LIN {X 0,Y 291.529,Z 647.486,A -85,B 0,C 180,E1 -16988.801,E2 -16988.801} C_VEL
LIN {X 0,Y 290.055,Z 656.21,A -85,B 0,C 180,E1 -16989.986,E2 -16989.986} C_VEL
LIN {X 0,Y 288.759,Z 663.631,A -85,B 0,C 180,E1 -16991.187,E2 -16991.187} C_VEL
LIN {X 0,Y 287.31,Z 672.431,A -85,B 0,C 180,E1 -16992.93,E2 -16992.93} C_VEL
LIN {X 0,Y 286.152,Z 678.42,A -85,B 0,C 180,E1 -16994.326,E2 -16994.326} C_VEL
LIN {X 0,Y 284.969,Z 684.732,A -85,B 0,C 180,E1 -16996.087,E2 -16996.087} C_VEL
LIN {X 0,Y 283.972,Z 690.005,A -85,B 0,C 180,E1 -16997.856,E2 -16997.856} C_VEL
LIN {X 0,Y 283.192,Z 695.101,A -85,B 0,C 180,E1 -16999.996,E2 -16999.996} C_VEL
LIN {X 0,Y 282.682,Z 699.069,A -85,B 0,C 180,E1 -17002.141,E2 -17002.141} C_VEL
LIN {X 0,Y 282.337,Z 702.443,A -85,B 0,C 180,E1 -17004.694,E2 -17004.694} C_VEL
LIN {X 0,Y 282.309,Z 703.508,A -85,B 0,C 180,E1 -17005.717,E2 -17005.717} C_VEL
LIN {X 0,Y 282.334,Z 705.035,A -85,B 0,C 180,E1 -17008.574,E2 -17008.574} C_VEL
LIN {X 0,Y 282.347,Z 705.315,A -85,B 0,C 180,E1 -17010,E2 -17010} C_VEL
LIN {X 0,Y 282.339,Z 704.439,A -85,B 0,C 180,E1 -17012.854,E2 -17012.854} C_VEL
LIN {X 0,Y 282.309,Z 703.508,A -85,B 0,C 180,E1 -17014.283,E2 -17014.283} C_VEL
LIN {X 0,Y 282.523,Z 700.157,A -85,B 0,C 180,E1 -17017.145,E2 -17017.145} C_VEL
LIN {X 0,Y 282.991,Z 696.53,A -85,B 0,C 180,E1 -17019.29,E2 -17019.29} C_VEL
LIN {X 0,Y 283.711,Z 691.797,A -85,B 0,C 180,E1 -17021.43,E2 -17021.43} C_VEL
LIN {X 0,Y 284.732,Z 685.823,A -85,B 0,C 180,E1 -17023.561,E2 -17023.561} C_VEL
LIN {X 0,Y 285.91,Z 679.733,A -85,B 0,C 180,E1 -17025.322,E2 -17025.322} C_VEL
LIN {X 0,Y 287.02,Z 673.992,A -85,B 0,C 180,E1 -17026.721,E2 -17026.721} C_VEL
LIN {X 0,Y 288.238,Z 667.091,A -85,B 0,C 180,E1 -17028.16,E2 -17028.16} C_VEL
LIN {X 0,Y 289.495,Z 659.505,A -85,B 0,C 180,E1 -17029.5,E2 -17029.5} C_VEL
LIN {X 0,Y 290.886,Z 651.424,A -85,B 0,C 180,E1 -17030.692,E2 -17030.692} C_VEL
LIN {X 0,Y 292.442,Z 641.666,A -85,B 0,C 180,E1 -17031.869,E2 -17031.869} C_VEL
LIN {X 0,Y 293.596,Z 633.277,A -85,B 0,C 180,E1 -17032.705,E2 -17032.705} C_VEL
LIN {X 0,Y 294.808,Z 622.772,A -85,B 0,C 180,E1 -17033.535,E2 -17033.535} C_VEL
LIN {X 0,Y 295.738,Z 612.44,A -85,B 0,C 180,E1 -17034.154,E2 -17034.154} C_VEL
LIN {X 0,Y 296.591,Z 601.726,A -85,B 0,C 180,E1 -17034.592,E2 -17034.592} C_VEL
LIN {X 0,Y 297.298,Z 578.95,A -85,B 0,C 180,E1 -17035.183,E2 -17035.183} C_VEL
LIN {X 0,Y 298.186,Z 540.495,A -85,B 0,C 180,E1 -17036.108,E2 -17036.108} C_VEL
LIN {X 0,Y 294.791,Z 520.737,A -85,B 0,C 180,E1 -17036.956,E2 -17036.956} C_VEL
LIN {X 0,Y 290.227,Z 500.059,A -85,B 0,C 180,E1 -17037.976,E2 -17037.976} C_VEL
LIN {X 0,Y 288.063,Z 494.317,A -85,B 0,C 180,E1 -17038.404,E2 -17038.404} C_VEL
LIN {X 0,Y 287.664,Z 492.009,A -85,B 0,C 180,E1 -17039.25,E2 -17039.25} C_VEL
LIN {X 0,Y 286.155,Z 484.135,A -85,B 0,C 180,E1 -17042.705,E2 -17042.705} C_VEL
LIN {X 0,Y 284.354,Z 475.643,A -85,B 0,C 180,E1 -17046.602,E2 -17046.602} C_VEL
LIN {X 0,Y 284.259,Z 475.55,A -85,B 0,C 180,E1 -17050.002,E2 -17050.002} C_VEL
LIN {X 0,Y 284.237,Z 475.58,A -85,B 0,C 180,E1 -17054.186,E2 -17054.186} C_VEL
LIN {X 0,Y 284.242,Z 475.579,A -85,B 0,C 180,E1 -17058.117,E2 -17058.117} C_VEL
LIN {X 0,Y 284.297,Z 475.566,A -85,B 0,C 180,E1 -17061.827,E2 -17061.827} C_VEL
LIN {X 0,Y 284.309,Z 475.551,A -85,B 0,C 180,E1 -17065.349,E2 -17065.349} C_VEL
LIN {X 0,Y 284.287,Z 475.573,A -85,B 0,C 180,E1 -17068.723,E2 -17068.723} C_VEL
LIN {X 0,Y 284.275,Z 475.553,A -85,B 0,C 180,E1 -17071.981,E2 -17071.981} C_VEL
LIN {X 0,Y 284.293,Z 475.566,A -85,B 0,C 180,E1 -17076.158,E2 -17076.158} C_VEL
LIN {X 0,Y 284.334,Z 475.543,A -85,B 0,C 180,E1 -17079.926,E2 -17079.926} C_VEL
LIN {X 0,Y 284.419,Z 475.547,A -85,B 0,C 180,E1 -17084.51,E2 -17084.51} C_VEL
LIN {X 0,Y 284.45,Z 475.533,A -85,B 0,C 180,E1 -17088.598,E2 -17088.598} C_VEL
LIN {X 0,Y 284.578,Z 475.499,A -85,B 0,C 180,E1 -17091.477,E2 -17091.477} C_VEL
LIN {X 0,Y 284.562,Z 475.535,A -85,B 0,C 180,E1 -17094.328,E2 -17094.328} C_VEL
LIN {X 0,Y 284.832,Z 475.483,A -85,B 0,C 180,E1 -17098.584,E2 -17098.584} C_VEL
LIN {X 0,Y 284.831,Z 475.469,A -85,B 0,C 180,E1 -17101.412,E2 -17101.412} C_VEL
LIN {X 0,Y 284.636,Z 475.523,A -85,B 0,C 180,E1 -17107.089,E2 -17107.089} C_VEL
LIN {X 0,Y 284.508,Z 475.507,A -85,B 0,C 180,E1 -17109.955,E2 -17109.955} C_VEL
LIN {X 0,Y 284.427,Z 475.557,A -85,B 0,C 180,E1 -17114.303,E2 -17114.303} C_VEL
LIN {X 0,Y 284.305,Z 475.536,A -85,B 0,C 180,E1 -17118.743,E2 -17118.743} C_VEL
LIN {X 0,Y 284.288,Z 475.562,A -85,B 0,C 180,E1 -17121.764,E2 -17121.764} C_VEL
LIN {X 0,Y 284.28,Z 475.569,A -85,B 0,C 180,E1 -17124.849,E2 -17124.849} C_VEL
LIN {X 0,Y 284.255,Z 475.55,A -85,B 0,C 180,E1 -17128.016,E2 -17128.016} C_VEL
LIN {X 0,Y 284.269,Z 475.576,A -85,B 0,C 180,E1 -17131.274,E2 -17131.274} C_VEL
LIN {X 0,Y 284.326,Z 475.549,A -85,B 0,C 180,E1 -17135.345,E2 -17135.345} C_VEL
LIN {X 0,Y 284.253,Z 475.578,A -85,B 0,C 180,E1 -17138.175,E2 -17138.175} C_VEL
LIN {X 0,Y 284.224,Z 475.571,A -85,B 0,C 180,E1 -17142.115,E2 -17142.115} C_VEL
LIN {X 0,Y 284.223,Z 475.543,A -85,B 0,C 180,E1 -17146.184,E2 -17146.184} C_VEL
LIN {X 0,Y 284.243,Z 475.546,A -85,B 0,C 180,E1 -17150.035,E2 -17150.035} C_VEL
LIN {X 0,Y 284.306,Z 475.551,A -85,B 0,C 180,E1 -17153.611,E2 -17153.611} C_VEL
LIN {X 0,Y 284.293,Z 475.554,A -85,B 0,C 180,E1 -17157.189,E2 -17157.189} C_VEL
LIN {X 0,Y 284.294,Z 475.725,A -85,B 0,C 180,E1 -17160.852,E2 -17160.852} C_VEL
LIN {X 0,Y 284.519,Z 476.73,A -85,B 0,C 180,E1 -17161.125,E2 -17161.125} C_VEL
LIN {X 0,Y 292.878,Z 492.327,A -85,B 0,C 180,E1 -17162.476,E2 -17162.476} C_VEL
LIN {X 0,Y 300.917,Z 503.502,A -85,B 0,C 180,E1 -17163.57,E2 -17163.57} C_VEL
LIN {X 0,Y 308.987,Z 512.535,A -85,B 0,C 180,E1 -17164.628,E2 -17164.628} C_VEL
LIN {X 0,Y 315.644,Z 519.573,A -85,B 0,C 180,E1 -17165.615,E2 -17165.615} C_VEL
LIN {X 0,Y 321.421,Z 525.437,A -85,B 0,C 180,E1 -17166.558,E2 -17166.558} C_VEL
LIN {X 0,Y 328.657,Z 532.455,A -85,B 0,C 180,E1 -17167.889,E2 -17167.889} C_VEL
LIN {X 0,Y 335.557,Z 538.982,A -85,B 0,C 180,E1 -17169.296,E2 -17169.296} C_VEL
LIN {X 0,Y 343.686,Z 546.102,A -85,B 0,C 180,E1 -17171.087,E2 -17171.087} C_VEL
LIN {X 0,Y 348.971,Z 550.286,A -85,B 0,C 180,E1 -17172.362,E2 -17172.362} C_VEL
LIN {X 0,Y 354.495,Z 554.841,A -85,B 0,C 180,E1 -17173.83,E2 -17173.83} C_VEL
LIN {X 0,Y 358.656,Z 557.939,A -85,B 0,C 180,E1 -17175.02,E2 -17175.02} C_VEL
LIN {X 0,Y 363.351,Z 561.774,A -85,B 0,C 180,E1 -17176.526,E2 -17176.526} C_VEL
LIN {X 0,Y 367.654,Z 564.654,A -85,B 0,C 180,E1 -17178.042,E2 -17178.042} C_VEL
LIN {X 0,Y 370.229,Z 566.282,A -85,B 0,C 180,E1 -17179.057,E2 -17179.057} C_VEL
LIN {X 0,Y 373.801,Z 569.424,A -85,B 0,C 180,E1 -17180.707,E2 -17180.707} C_VEL
LIN {X 0,Y 376.944,Z 571.542,A -85,B 0,C 180,E1 -17182.409,E2 -17182.409} C_VEL
LIN {X 0,Y 379.734,Z 573.137,A -85,B 0,C 180,E1 -17184.311,E2 -17184.311} C_VEL
LIN {X 0,Y 381.683,Z 573.837,A -85,B 0,C 180,E1 -17186.144,E2 -17186.144} C_VEL
LIN {X 0,Y 382.823,Z 574.391,A -85,B 0,C 180,E1 -17187.896,E2 -17187.896} C_VEL
LIN {X 0,Y 383.197,Z 574.651,A -85,B 0,C 180,E1 -17188.949,E2 -17188.949} C_VEL
LIN {X 0,Y 383.338,Z 574.609,A -85,B 0,C 180,E1 -17190,E2 -17190} C_VEL
LIN {X 0,Y 382.956,Z 574.451,A -85,B 0,C 180,E1 -17191.84,E2 -17191.84} C_VEL
LIN {X 0,Y 381.682,Z 573.849,A -85,B 0,C 180,E1 -17193.854,E2 -17193.854} C_VEL
LIN {X 0,Y 379.685,Z 573.06,A -85,B 0,C 180,E1 -17195.732,E2 -17195.732} C_VEL
LIN {X 0,Y 376.692,Z 571.448,A -85,B 0,C 180,E1 -17197.73,E2 -17197.73} C_VEL
LIN {X 0,Y 373.535,Z 569.224,A -85,B 0,C 180,E1 -17199.421,E2 -17199.421} C_VEL
LIN {X 0,Y 369.66,Z 565.748,A -85,B 0,C 180,E1 -17201.184,E2 -17201.184} C_VEL
LIN {X 0,Y 365.169,Z 563.042,A -85,B 0,C 180,E1 -17202.852,E2 -17202.852} C_VEL
LIN {X 0,Y 360.317,Z 559.407,A -85,B 0,C 180,E1 -17204.458,E2 -17204.458} C_VEL
LIN {X 0,Y 356.054,Z 555.938,A -85,B 0,C 180,E1 -17205.739,E2 -17205.739} C_VEL
LIN {X 0,Y 350.445,Z 551.606,A -85,B 0,C 180,E1 -17207.252,E2 -17207.252} C_VEL
LIN {X 0,Y 345.679,Z 547.625,A -85,B 0,C 180,E1 -17208.44,E2 -17208.44} C_VEL
LIN {X 0,Y 339.714,Z 542.632,A -85,B 0,C 180,E1 -17209.815,E2 -17209.815} C_VEL
LIN {X 0,Y 331.377,Z 535.125,A -85,B 0,C 180,E1 -17211.572,E2 -17211.572} C_VEL
LIN {X 0,Y 323.219,Z 527.28,A -85,B 0,C 180,E1 -17213.117,E2 -17213.117} C_VEL
LIN {X 0,Y 316.382,Z 520.409,A -85,B 0,C 180,E1 -17214.265,E2 -17214.265} C_VEL
LIN {X 0,Y 309.394,Z 512.951,A -85,B 0,C 180,E1 -17215.317,E2 -17215.317} C_VEL
LIN {X 0,Y 301.321,Z 504.014,A -85,B 0,C 180,E1 -17216.378,E2 -17216.378} C_VEL
LIN {X 0,Y 293.463,Z 493.195,A -85,B 0,C 180,E1 -17217.44,E2 -17217.44} C_VEL
LIN {X 0,Y 287.712,Z 482.971,A -85,B 0,C 180,E1 -17218.326,E2 -17218.326} C_VEL
LIN {X 0,Y 284.463,Z 476.5,A -85,B 0,C 180,E1 -17218.907,E2 -17218.907} C_VEL
LIN {X 0,Y 284.265,Z 475.622,A -85,B 0,C 180,E1 -17219.234,E2 -17219.234} C_VEL
LIN {X 0,Y 284.291,Z 475.552,A -85,B 0,C 180,E1 -17222.947,E2 -17222.947} C_VEL
LIN {X 0,Y 284.306,Z 475.551,A -85,B 0,C 180,E1 -17226.389,E2 -17226.389} C_VEL
LIN {X 0,Y 284.242,Z 475.545,A -85,B 0,C 180,E1 -17230.005,E2 -17230.005} C_VEL
LIN {X 0,Y 284.22,Z 475.552,A -85,B 0,C 180,E1 -17234.189,E2 -17234.189} C_VEL
LIN {X 0,Y 284.227,Z 475.569,A -85,B 0,C 180,E1 -17238.12,E2 -17238.12} C_VEL
LIN {X 0,Y 284.271,Z 475.577,A -85,B 0,C 180,E1 -17242.291,E2 -17242.291} C_VEL
LIN {X 0,Y 284.296,Z 475.549,A -85,B 0,C 180,E1 -17245.352,E2 -17245.352} C_VEL
LIN {X 0,Y 284.269,Z 475.576,A -85,B 0,C 180,E1 -17248.726,E2 -17248.726} C_VEL
LIN {X 0,Y 284.255,Z 475.55,A -85,B 0,C 180,E1 -17251.984,E2 -17251.984} C_VEL
LIN {X 0,Y 284.29,Z 475.575,A -85,B 0,C 180,E1 -17256.16,E2 -17256.16} C_VEL
LIN {X 0,Y 284.326,Z 475.536,A -85,B 0,C 180,E1 -17259.93,E2 -17259.93} C_VEL
LIN {X 0,Y 284.408,Z 475.558,A -85,B 0,C 180,E1 -17264.519,E2 -17264.519} C_VEL
LIN {X 0,Y 284.456,Z 475.522,A -85,B 0,C 180,E1 -17268.603,E2 -17268.603} C_VEL
LIN {X 0,Y 284.603,Z 475.509,A -85,B 0,C 180,E1 -17271.482,E2 -17271.482} C_VEL
LIN {X 0,Y 284.56,Z 475.539,A -85,B 0,C 180,E1 -17274.333,E2 -17274.333} C_VEL
LIN {X 0,Y 284.831,Z 475.469,A -85,B 0,C 180,E1 -17278.588,E2 -17278.588} C_VEL
LIN {X 0,Y 284.832,Z 475.483,A -85,B 0,C 180,E1 -17281.416,E2 -17281.416} C_VEL
LIN {X 0,Y 284.634,Z 475.511,A -85,B 0,C 180,E1 -17287.094,E2 -17287.094} C_VEL
LIN {X 0,Y 284.507,Z 475.507,A -85,B 0,C 180,E1 -17289.959,E2 -17289.959} C_VEL
LIN {X 0,Y 284.404,Z 475.555,A -85,B 0,C 180,E1 -17294.309,E2 -17294.309} C_VEL
LIN {X 0,Y 284.326,Z 475.538,A -85,B 0,C 180,E1 -17297.257,E2 -17297.257} C_VEL
LIN {X 0,Y 284.327,Z 475.542,A -85,B 0,C 180,E1 -17299.986,E2 -17299.986} C_VEL
LIN {X 0,Y 283.715,Z 475.635,A -85,B 0,C 180,E1 -17301.168,E2 -17301.168} C_VEL
LIN {X 0,Y 280.834,Z 476,A -85,B 0,C 180,E1 -17303.093,E2 -17303.093} C_VEL
LIN {X 0,Y 278.355,Z 476.3,A -85,B 0,C 180,E1 -17304.657,E2 -17304.657} C_VEL
LIN {X 0,Y 277.296,Z 476.415,A -85,B 0,C 180,E1 -17305.871,E2 -17305.871} C_VEL
LIN {X 0,Y 277.216,Z 476.422,A -85,B 0,C 180,E1 -17306.283,E2 -17306.283} C_VEL
LIN {X 0,Y 277.25,Z 476.449,A -85,B 0,C 180,E1 -17310.475,E2 -17310.475} C_VEL
LIN {X 0,Y 277.248,Z 476.426,A -85,B 0,C 180,E1 -17313.898,E2 -17313.898} C_VEL
LIN {X 0,Y 277.253,Z 476.45,A -85,B 0,C 180,E1 -17317.474,E2 -17317.474} C_VEL
LIN {X 0,Y 277.187,Z 476.454,A -85,B 0,C 180,E1 -17321.243,E2 -17321.243} C_VEL
LIN {X 0,Y 277.177,Z 476.456,A -85,B 0,C 180,E1 -17325.234,E2 -17325.234} C_VEL
LIN {X 0,Y 277.18,Z 476.428,A -85,B 0,C 180,E1 -17328.759,E2 -17328.759} C_VEL
LIN {X 0,Y 277.303,Z 476.579,A -85,B 0,C 180,E1 -17332.849,E2 -17332.849} C_VEL
LIN {X 0,Y 278.891,Z 483.907,A -85,B 0,C 180,E1 -17336.331,E2 -17336.331} C_VEL
LIN {X 0,Y 280.441,Z 491.786,A -85,B 0,C 180,E1 -17339.92,E2 -17339.92} C_VEL
LIN {X 0,Y 280.846,Z 494.095,A -85,B 0,C 180,E1 -17340.795,E2 -17340.795} C_VEL
LIN {X 0,Y 284.507,Z 503.564,A -85,B 0,C 180,E1 -17341.514,E2 -17341.514} C_VEL
LIN {X 0,Y 289.339,Z 526.516,A -85,B 0,C 180,E1 -17342.657,E2 -17342.657} C_VEL
LIN {X 0,Y 291.813,Z 541.536,A -85,B 0,C 180,E1 -17343.311,E2 -17343.311} C_VEL
LIN {X 0,Y 290.242,Z 600.213,A -85,B 0,C 180,E1 -17344.785,E2 -17344.785} C_VEL
LIN {X 0,Y 289.578,Z 609.664,A -85,B 0,C 180,E1 -17345.155,E2 -17345.155} C_VEL
LIN {X 0,Y 288.729,Z 618.789,A -85,B 0,C 180,E1 -17345.652,E2 -17345.652} C_VEL
LIN {X 0,Y 287.555,Z 629.145,A -85,B 0,C 180,E1 -17346.409,E2 -17346.409} C_VEL
LIN {X 0,Y 286.303,Z 638.289,A -85,B 0,C 180,E1 -17347.256,E2 -17347.256} C_VEL
LIN {X 0,Y 284.911,Z 647.289,A -85,B 0,C 180,E1 -17348.284,E2 -17348.284} C_VEL
LIN {X 0,Y 283.4,Z 656.014,A -85,B 0,C 180,E1 -17349.496,E2 -17349.496} C_VEL
LIN {X 0,Y 282.017,Z 663.434,A -85,B 0,C 180,E1 -17350.72,E2 -17350.72} C_VEL
LIN {X 0,Y 280.743,Z 671.058,A -85,B 0,C 180,E1 -17352.235,E2 -17352.235} C_VEL
LIN {X 0,Y 279.28,Z 678.223,A -85,B 0,C 180,E1 -17353.93,E2 -17353.93} C_VEL
LIN {X 0,Y 278.035,Z 684.534,A -85,B 0,C 180,E1 -17355.732,E2 -17355.732} C_VEL
LIN {X 0,Y 276.993,Z 689.807,A -85,B 0,C 180,E1 -17357.546,E2 -17357.546} C_VEL
LIN {X 0,Y 276.181,Z 694.905,A -85,B 0,C 180,E1 -17359.739,E2 -17359.739} C_VEL
LIN {X 0,Y 275.612,Z 698.871,A -85,B 0,C 180,E1 -17361.938,E2 -17361.938} C_VEL
LIN {X 0,Y 275.23,Z 702.504,A -85,B 0,C 180,E1 -17364.804,E2 -17364.804} C_VEL
LIN {X 0,Y 275.248,Z 704.243,A -85,B 0,C 180,E1 -17367.073,E2 -17367.073} C_VEL
LIN {X 0,Y 275.27,Z 705.119,A -85,B 0,C 180,E1 -17370,E2 -17370} C_VEL
LIN {X 0,Y 275.248,Z 704.243,A -85,B 0,C 180,E1 -17372.927,E2 -17372.927} C_VEL
LIN {X 0,Y 275.244,Z 702.472,A -85,B 0,C 180,E1 -17375.227,E2 -17375.227} C_VEL
LIN {X 0,Y 275.612,Z 698.871,A -85,B 0,C 180,E1 -17378.062,E2 -17378.062} C_VEL
LIN {X 0,Y 276.181,Z 694.905,A -85,B 0,C 180,E1 -17380.261,E2 -17380.261} C_VEL
LIN {X 0,Y 276.993,Z 689.807,A -85,B 0,C 180,E1 -17382.454,E2 -17382.454} C_VEL
LIN {X 0,Y 278.544,Z 682.159,A -85,B 0,C 180,E1 -17384.988,E2 -17384.988} C_VEL
LIN {X 0,Y 279.885,Z 675.355,A -85,B 0,C 180,E1 -17386.784,E2 -17386.784} C_VEL
LIN {X 0,Y 281.403,Z 667.259,A -85,B 0,C 180,E1 -17388.543,E2 -17388.543} C_VEL
LIN {X 0,Y 282.788,Z 659.309,A -85,B 0,C 180,E1 -17389.982,E2 -17389.982} C_VEL
LIN {X 0,Y 284.242,Z 651.227,A -85,B 0,C 180,E1 -17391.199,E2 -17391.199} C_VEL
LIN {X 0,Y 285.866,Z 641.469,A -85,B 0,C 180,E1 -17392.399,E2 -17392.399} C_VEL
LIN {X 0,Y 287.075,Z 633.081,A -85,B 0,C 180,E1 -17393.251,E2 -17393.251} C_VEL
LIN {X 0,Y 288.301,Z 622.575,A -85,B 0,C 180,E1 -17394.099,E2 -17394.099} C_VEL
LIN {X 0,Y 289.275,Z 612.244,A -85,B 0,C 180,E1 -17394.729,E2 -17394.729} C_VEL
LIN {X 0,Y 290.168,Z 601.53,A -85,B 0,C 180,E1 -17395.174,E2 -17395.174} C_VEL
LIN {X 0,Y 290.911,Z 577.482,A -85,B 0,C 180,E1 -17395.81,E2 -17395.81} C_VEL
LIN {X 0,Y 291.813,Z 541.474,A -85,B 0,C 180,E1 -17396.691,E2 -17396.691} C_VEL
LIN {X 0,Y 288.218,Z 520.714,A -85,B 0,C 180,E1 -17397.617,E2 -17397.617} C_VEL
LIN {X 0,Y 284.223,Z 502.691,A -85,B 0,C 180,E1 -17398.541,E2 -17398.541} C_VEL
LIN {X 0,Y 280.863,Z 494.04,A -85,B 0,C 180,E1 -17399.209,E2 -17399.209} C_VEL
LIN {X 0,Y 279.881,Z 488.936,A -85,B 0,C 180,E1 -17401.374,E2 -17401.374} C_VEL
LIN {X 0,Y 278.24,Z 480.908,A -85,B 0,C 180,E1 -17405.073,E2 -17405.073} C_VEL
LIN {X 0,Y 277.292,Z 476.505,A -85,B 0,C 180,E1 -17407.257,E2 -17407.257} C_VEL
LIN {X 0,Y 277.179,Z 476.428,A -85,B 0,C 180,E1 -17411.242,E2 -17411.242} C_VEL
LIN {X 0,Y 277.177,Z 476.451,A -85,B 0,C 180,E1 -17415.231,E2 -17415.231} C_VEL
LIN {X 0,Y 277.187,Z 476.454,A -85,B 0,C 180,E1 -17418.757,E2 -17418.757} C_VEL
LIN {X 0,Y 277.253,Z 476.45,A -85,B 0,C 180,E1 -17422.526,E2 -17422.526} C_VEL
LIN {X 0,Y 277.248,Z 476.426,A -85,B 0,C 180,E1 -17426.102,E2 -17426.102} C_VEL
LIN {X 0,Y 277.264,Z 476.448,A -85,B 0,C 180,E1 -17429.537,E2 -17429.537} C_VEL
LIN {X 0,Y 277.256,Z 476.418,A -85,B 0,C 180,E1 -17432.851,E2 -17432.851} C_VEL
LIN {X 0,Y 277.256,Z 476.441,A -85,B 0,C 180,E1 -17436.071,E2 -17436.071} C_VEL
LIN {X 0,Y 277.271,Z 476.425,A -85,B 0,C 180,E1 -17439.69,E2 -17439.69} C_VEL
LIN {X 0,Y 277.369,Z 476.423,A -85,B 0,C 180,E1 -17444.331,E2 -17444.331} C_VEL
LIN {X 0,Y 277.399,Z 476.413,A -85,B 0,C 180,E1 -17448.304,E2 -17448.304} C_VEL
LIN {X 0,Y 277.549,Z 476.372,A -85,B 0,C 180,E1 -17451.259,E2 -17451.259} C_VEL
LIN {X 0,Y 277.533,Z 476.408,A -85,B 0,C 180,E1 -17454.184,E2 -17454.184} C_VEL
LIN {X 0,Y 277.799,Z 476.359,A -85,B 0,C 180,E1 -17458.548,E2 -17458.548} C_VEL
LIN {X 0,Y 277.798,Z 476.345,A -85,B 0,C 180,E1 -17461.447,E2 -17461.447} C_VEL
LIN {X 0,Y 277.594,Z 476.397,A -85,B 0,C 180,E1 -17467.27,E2 -17467.27} C_VEL
LIN {X 0,Y 277.448,Z 476.385,A -85,B 0,C 180,E1 -17470.211,E2 -17470.211} C_VEL
LIN {X 0,Y 277.374,Z 476.434,A -85,B 0,C 180,E1 -17474.675,E2 -17474.675} C_VEL
LIN {X 0,Y 277.266,Z 476.411,A -85,B 0,C 180,E1 -17479.237,E2 -17479.237} C_VEL
LIN {X 0,Y 277.252,Z 476.451,A -85,B 0,C 180,E1 -17483.925,E2 -17483.925} C_VEL
LIN {X 0,Y 277.229,Z 476.423,A -85,B 0,C 180,E1 -17487.468,E2 -17487.468} C_VEL
LIN {X 0,Y 277.219,Z 476.454,A -85,B 0,C 180,E1 -17490.464,E2 -17490.464} C_VEL
LIN {X 0,Y 277.236,Z 476.431,A -85,B 0,C 180,E1 -17493.894,E2 -17493.894} C_VEL
LIN {X 0,Y 277.222,Z 476.453,A -85,B 0,C 180,E1 -17497.473,E2 -17497.473} C_VEL
LIN {X 0,Y 277.165,Z 476.443,A -85,B 0,C 180,E1 -17501.241,E2 -17501.241} C_VEL
LIN {X 0,Y 277.161,Z 476.441,A -85,B 0,C 180,E1 -17505.231,E2 -17505.231} C_VEL
LIN {X 0,Y 277.162,Z 476.416,A -85,B 0,C 180,E1 -17509.522,E2 -17509.522} C_VEL
LIN {X 0,Y 277.236,Z 476.451,A -85,B 0,C 180,E1 -17512.526,E2 -17512.526} C_VEL
LIN {X 0,Y 277.233,Z 476.418,A -85,B 0,C 180,E1 -17516.103,E2 -17516.103} C_VEL
LIN {X 0,Y 277.262,Z 476.562,A -85,B 0,C 180,E1 -17520.053,E2 -17520.053} C_VEL
LIN {X 0,Y 277.479,Z 477.493,A -85,B 0,C 180,E1 -17520.332,E2 -17520.332} C_VEL
LIN {X 0,Y 287.526,Z 496.408,A -85,B 0,C 180,E1 -17522.028,E2 -17522.028} C_VEL
LIN {X 0,Y 295.653,Z 507.858,A -85,B 0,C 180,E1 -17523.174,E2 -17523.174} C_VEL
LIN {X 0,Y 304.765,Z 518.008,A -85,B 0,C 180,E1 -17524.326,E2 -17524.326} C_VEL
LIN {X 0,Y 311.377,Z 524.867,A -85,B 0,C 180,E1 -17525.238,E2 -17525.238} C_VEL
LIN {X 0,Y 317.729,Z 531.19,A -85,B 0,C 180,E1 -17526.208,E2 -17526.208} C_VEL
LIN {X 0,Y 324.549,Z 537.729,A -85,B 0,C 180,E1 -17527.392,E2 -17527.392} C_VEL
LIN {X 0,Y 332.413,Z 544.955,A -85,B 0,C 180,E1 -17528.906,E2 -17528.906} C_VEL
LIN {X 0,Y 340.777,Z 552.181,A -85,B 0,C 180,E1 -17530.701,E2 -17530.701} C_VEL
LIN {X 0,Y 346.561,Z 556.69,A -85,B 0,C 180,E1 -17532.049,E2 -17532.049} C_VEL
LIN {X 0,Y 352.505,Z 561.473,A -85,B 0,C 180,E1 -17533.576,E2 -17533.576} C_VEL
LIN {X 0,Y 356.962,Z 564.812,A -85,B 0,C 180,E1 -17534.828,E2 -17534.828} C_VEL
LIN {X 0,Y 362.405,Z 569.047,A -85,B 0,C 180,E1 -17536.543,E2 -17536.543} C_VEL
LIN {X 0,Y 366.729,Z 571.78,A -85,B 0,C 180,E1 -17538.054,E2 -17538.054} C_VEL
LIN {X 0,Y 368.799,Z 573.161,A -85,B 0,C 180,E1 -17538.863,E2 -17538.863} C_VEL
LIN {X 0,Y 372.649,Z 576.424,A -85,B 0,C 180,E1 -17540.599,E2 -17540.599} C_VEL
LIN {X 0,Y 375.854,Z 578.514,A -85,B 0,C 180,E1 -17542.303,E2 -17542.303} C_VEL
LIN {X 0,Y 378.833,Z 580.178,A -85,B 0,C 180,E1 -17544.298,E2 -17544.298} C_VEL
LIN {X 0,Y 380.509,Z 580.767,A -85,B 0,C 180,E1 -17545.819,E2 -17545.819} C_VEL
LIN {X 0,Y 381.68,Z 581.241,A -85,B 0,C 180,E1 -17547.348,E2 -17547.348} C_VEL
LIN {X 0,Y 382.335,Z 581.681,A -85,B 0,C 180,E1 -17548.947,E2 -17548.947} C_VEL
LIN {X 0,Y 382.475,Z 581.643,A -85,B 0,C 180,E1 -17550,E2 -17550} C_VEL
LIN {X 0,Y 382.088,Z 581.506,A -85,B 0,C 180,E1 -17551.845,E2 -17551.845} C_VEL
LIN {X 0,Y 381.088,Z 580.947,A -85,B 0,C 180,E1 -17553.516,E2 -17553.516} C_VEL
LIN {X 0,Y 379.001,Z 580.232,A -85,B 0,C 180,E1 -17555.564,E2 -17555.564} C_VEL
LIN {X 0,Y 376.177,Z 578.691,A -85,B 0,C 180,E1 -17557.515,E2 -17557.515} C_VEL
LIN {X 0,Y 372.74,Z 576.454,A -85,B 0,C 180,E1 -17559.359,E2 -17559.359} C_VEL
LIN {X 0,Y 368.99,Z 573.319,A -85,B 0,C 180,E1 -17561.059,E2 -17561.059} C_VEL
LIN {X 0,Y 366.925,Z 571.902,A -85,B 0,C 180,E1 -17561.873,E2 -17561.873} C_VEL
LIN {X 0,Y 362.063,Z 568.81,A -85,B 0,C 180,E1 -17563.576,E2 -17563.576} C_VEL
LIN {X 0,Y 356.159,Z 564.11,A -85,B 0,C 180,E1 -17565.413,E2 -17565.413} C_VEL
LIN {X 0,Y 349.393,Z 559.104,A -85,B 0,C 180,E1 -17567.233,E2 -17567.233} C_VEL
LIN {X 0,Y 342.736,Z 553.647,A -85,B 0,C 180,E1 -17568.863,E2 -17568.863} C_VEL
LIN {X 0,Y 336.716,Z 548.656,A -85,B 0,C 180,E1 -17570.199,E2 -17570.199} C_VEL
LIN {X 0,Y 328.333,Z 541.273,A -85,B 0,C 180,E1 -17571.903,E2 -17571.903} C_VEL
LIN {X 0,Y 319.945,Z 533.412,A -85,B 0,C 180,E1 -17573.419,E2 -17573.419} C_VEL
LIN {X 0,Y 312.232,Z 525.808,A -85,B 0,C 180,E1 -17574.636,E2 -17574.636} C_VEL
LIN {X 0,Y 304.264,Z 517.527,A -85,B 0,C 180,E1 -17575.738,E2 -17575.738} C_VEL
LIN {X 0,Y 294.748,Z 506.641,A -85,B 0,C 180,E1 -17576.948,E2 -17576.948} C_VEL
LIN {X 0,Y 287.309,Z 496.046,A -85,B 0,C 180,E1 -17578.006,E2 -17578.006} C_VEL
LIN {X 0,Y 277.478,Z 477.492,A -85,B 0,C 180,E1 -17579.667,E2 -17579.667} C_VEL
LIN {X 0,Y 277.243,Z 476.498,A -85,B 0,C 180,E1 -17580.006,E2 -17580.006} C_VEL
LIN {X 0,Y 277.233,Z 476.418,A -85,B 0,C 180,E1 -17583.897,E2 -17583.897} C_VEL
LIN {X 0,Y 277.236,Z 476.451,A -85,B 0,C 180,E1 -17587.474,E2 -17587.474} C_VEL
LIN {X 0,Y 277.16,Z 476.407,A -85,B 0,C 180,E1 -17591.245,E2 -17591.245} C_VEL
LIN {X 0,Y 277.162,Z 476.451,A -85,B 0,C 180,E1 -17595.234,E2 -17595.234} C_VEL
LIN {X 0,Y 277.165,Z 476.443,A -85,B 0,C 180,E1 -17598.759,E2 -17598.759} C_VEL
LIN {X 0,Y 277.222,Z 476.453,A -85,B 0,C 180,E1 -17602.527,E2 -17602.527} C_VEL
LIN {X 0,Y 277.236,Z 476.431,A -85,B 0,C 180,E1 -17606.106,E2 -17606.106} C_VEL
LIN {X 0,Y 277.219,Z 476.454,A -85,B 0,C 180,E1 -17609.536,E2 -17609.536} C_VEL
LIN {X 0,Y 277.245,Z 476.421,A -85,B 0,C 180,E1 -17612.855,E2 -17612.855} C_VEL
LIN {X 0,Y 277.252,Z 476.451,A -85,B 0,C 180,E1 -17616.075,E2 -17616.075} C_VEL
LIN {X 0,Y 277.266,Z 476.411,A -85,B 0,C 180,E1 -17620.763,E2 -17620.763} C_VEL
LIN {X 0,Y 277.374,Z 476.434,A -85,B 0,C 180,E1 -17625.325,E2 -17625.325} C_VEL
LIN {X 0,Y 277.448,Z 476.385,A -85,B 0,C 180,E1 -17629.789,E2 -17629.789} C_VEL
LIN {X 0,Y 277.594,Z 476.397,A -85,B 0,C 180,E1 -17632.73,E2 -17632.73} C_VEL
LIN {X 0,Y 277.798,Z 476.345,A -85,B 0,C 180,E1 -17638.553,E2 -17638.553} C_VEL
LIN {X 0,Y 277.799,Z 476.359,A -85,B 0,C 180,E1 -17641.452,E2 -17641.452} C_VEL
LIN {X 0,Y 277.59,Z 476.384,A -85,B 0,C 180,E1 -17647.275,E2 -17647.275} C_VEL
LIN {X 0,Y 277.448,Z 476.387,A -85,B 0,C 180,E1 -17650.216,E2 -17650.216} C_VEL
LIN {X 0,Y 277.363,Z 476.43,A -85,B 0,C 180,E1 -17654.68,E2 -17654.68} C_VEL
LIN {X 0,Y 277.267,Z 476.413,A -85,B 0,C 180,E1 -17659.242,E2 -17659.242} C_VEL
LIN {X 0,Y 277.246,Z 476.448,A -85,B 0,C 180,E1 -17662.351,E2 -17662.351} C_VEL
LIN {X 0,Y 277.216,Z 476.422,A -85,B 0,C 180,E1 -17666.283,E2 -17666.283} C_VEL
LIN {X 0,Y 276.552,Z 476.511,A -85,B 0,C 180,E1 -17667.495,E2 -17667.495} C_VEL
LIN {X 0,Y 273.667,Z 476.891,A -85,B 0,C 180,E1 -17669.47,E2 -17669.47} C_VEL
LIN {X 0,Y 271.239,Z 477.197,A -85,B 0,C 180,E1 -17671.076,E2 -17671.076} C_VEL
LIN {X 0,Y 270.237,Z 477.311,A -85,B 0,C 180,E1 -17672.321,E2 -17672.321} C_VEL
LIN {X 0,Y 270.177,Z 477.311,A -85,B 0,C 180,E1 -17672.742,E2 -17672.742} C_VEL
LIN {X 0,Y 270.209,Z 477.326,A -85,B 0,C 180,E1 -17676.745,E2 -17676.745} C_VEL
LIN {X 0,Y 270.15,Z 477.323,A -85,B 0,C 180,E1 -17680.572,E2 -17680.572} C_VEL
LIN {X 0,Y 270.132,Z 477.328,A -85,B 0,C 180,E1 -17684.627,E2 -17684.627} C_VEL
LIN {X 0,Y 270.154,Z 477.317,A -85,B 0,C 180,E1 -17687.439,E2 -17687.439} C_VEL
LIN {X 0,Y 270.232,Z 477.429,A -85,B 0,C 180,E1 -17692.209,E2 -17692.209} C_VEL
LIN {X 0,Y 271.838,Z 484.771,A -85,B 0,C 180,E1 -17695.827,E2 -17695.827} C_VEL
LIN {X 0,Y 273.615,Z 493.673,A -85,B 0,C 180,E1 -17699.913,E2 -17699.913} C_VEL
LIN {X 0,Y 275.306,Z 498.06,A -85,B 0,C 180,E1 -17700.317,E2 -17700.317} C_VEL
LIN {X 0,Y 278.641,Z 506.366,A -85,B 0,C 180,E1 -17700.943,E2 -17700.943} C_VEL
LIN {X 0,Y 283.73,Z 531.197,A -85,B 0,C 180,E1 -17702.205,E2 -17702.205} C_VEL
LIN {X 0,Y 285.474,Z 543.231,A -85,B 0,C 180,E1 -17702.722,E2 -17702.722} C_VEL
LIN {X 0,Y 283.814,Z 600.023,A -85,B 0,C 180,E1 -17704.173,E2 -17704.173} C_VEL
LIN {X 0,Y 283.163,Z 609.468,A -85,B 0,C 180,E1 -17704.552,E2 -17704.552} C_VEL
LIN {X 0,Y 282.254,Z 618.592,A -85,B 0,C 180,E1 -17705.056,E2 -17705.056} C_VEL
LIN {X 0,Y 281.368,Z 626.982,A -85,B 0,C 180,E1 -17705.661,E2 -17705.661} C_VEL
LIN {X 0,Y 279.759,Z 638.092,A -85,B 0,C 180,E1 -17706.693,E2 -17706.693} C_VEL
LIN {X 0,Y 278.311,Z 647.093,A -85,B 0,C 180,E1 -17707.742,E2 -17707.742} C_VEL
LIN {X 0,Y 276.753,Z 655.818,A -85,B 0,C 180,E1 -17708.98,E2 -17708.98} C_VEL
LIN {X 0,Y 275.315,Z 663.237,A -85,B 0,C 180,E1 -17710.231,E2 -17710.231} C_VEL
LIN {X 0,Y 273.713,Z 672.037,A -85,B 0,C 180,E1 -17712.054,E2 -17712.054} C_VEL
LIN {X 0,Y 272.434,Z 678.026,A -85,B 0,C 180,E1 -17713.515,E2 -17713.515} C_VEL
LIN {X 0,Y 271.132,Z 684.337,A -85,B 0,C 180,E1 -17715.361,E2 -17715.361} C_VEL
LIN {X 0,Y 270.032,Z 689.61,A -85,B 0,C 180,E1 -17717.219,E2 -17717.219} C_VEL
LIN {X 0,Y 269.167,Z 694.708,A -85,B 0,C 180,E1 -17719.469,E2 -17719.469} C_VEL
LIN {X 0,Y 268.559,Z 698.674,A -85,B 0,C 180,E1 -17721.725,E2 -17721.725} C_VEL
LIN {X 0,Y 268.13,Z 702.553,A -85,B 0,C 180,E1 -17724.907,E2 -17724.907} C_VEL
LIN {X 0,Y 268.159,Z 704.046,A -85,B 0,C 180,E1 -17726.995,E2 -17726.995} C_VEL
LIN {X 0,Y 268.194,Z 704.924,A -85,B 0,C 180,E1 -17730,E2 -17730} C_VEL
LIN {X 0,Y 268.16,Z 704.046,A -85,B 0,C 180,E1 -17733.005,E2 -17733.005} C_VEL
LIN {X 0,Y 268.169,Z 702.457,A -85,B 0,C 180,E1 -17735.187,E2 -17735.187} C_VEL
LIN {X 0,Y 268.559,Z 698.674,A -85,B 0,C 180,E1 -17738.275,E2 -17738.275} C_VEL
LIN {X 0,Y 269.167,Z 694.708,A -85,B 0,C 180,E1 -17740.531,E2 -17740.531} C_VEL
LIN {X 0,Y 270.032,Z 689.61,A -85,B 0,C 180,E1 -17742.781,E2 -17742.781} C_VEL
LIN {X 0,Y 271.675,Z 681.963,A -85,B 0,C 180,E1 -17745.376,E2 -17745.376} C_VEL
LIN {X 0,Y 273.092,Z 675.159,A -85,B 0,C 180,E1 -17747.214,E2 -17747.214} C_VEL
LIN {X 0,Y 274.384,Z 668.599,A -85,B 0,C 180,E1 -17748.713,E2 -17748.713} C_VEL
LIN {X 0,Y 276.096,Z 659.111,A -85,B 0,C 180,E1 -17750.487,E2 -17750.487} C_VEL
LIN {X 0,Y 277.613,Z 651.03,A -85,B 0,C 180,E1 -17751.73,E2 -17751.73} C_VEL
LIN {X 0,Y 279.317,Z 641.273,A -85,B 0,C 180,E1 -17752.954,E2 -17752.954} C_VEL
LIN {X 0,Y 280.579,Z 632.885,A -85,B 0,C 180,E1 -17753.822,E2 -17753.822} C_VEL
LIN {X 0,Y 281.839,Z 622.379,A -85,B 0,C 180,E1 -17754.688,E2 -17754.688} C_VEL
LIN {X 0,Y 282.843,Z 612.048,A -85,B 0,C 180,E1 -17755.331,E2 -17755.331} C_VEL
LIN {X 0,Y 283.769,Z 601.334,A -85,B 0,C 180,E1 -17755.783,E2 -17755.783} C_VEL
LIN {X 0,Y 284.54,Z 577.424,A -85,B 0,C 180,E1 -17756.428,E2 -17756.428} C_VEL
LIN {X 0,Y 285.41,Z 541.956,A -85,B 0,C 180,E1 -17757.32,E2 -17757.32} C_VEL
LIN {X 0,Y 281.875,Z 521.759,A -85,B 0,C 180,E1 -17758.259,E2 -17758.259} C_VEL
LIN {X 0,Y 278.317,Z 505.345,A -85,B 0,C 180,E1 -17759.123,E2 -17759.123} C_VEL
LIN {X 0,Y 273.689,Z 494.043,A -85,B 0,C 180,E1 -17760.025,E2 -17760.025} C_VEL
LIN {X 0,Y 273.516,Z 493.194,A -85,B 0,C 180,E1 -17760.24,E2 -17760.24} C_VEL
LIN {X 0,Y 271.83,Z 484.779,A -85,B 0,C 180,E1 -17764.171,E2 -17764.171} C_VEL
LIN {X 0,Y 270.219,Z 477.402,A -85,B 0,C 180,E1 -17767.853,E2 -17767.853} C_VEL
LIN {X 0,Y 270.153,Z 477.316,A -85,B 0,C 180,E1 -17772.561,E2 -17772.561} C_VEL
LIN {X 0,Y 270.15,Z 477.328,A -85,B 0,C 180,E1 -17776.754,E2 -17776.754} C_VEL
LIN {X 0,Y 270.195,Z 477.319,A -85,B 0,C 180,E1 -17781.37,E2 -17781.37} C_VEL
LIN {X 0,Y 270.199,Z 477.309,A -85,B 0,C 180,E1 -17785.092,E2 -17785.092} C_VEL
LIN {X 0,Y 270.186,Z 477.328,A -85,B 0,C 180,E1 -17789.135,E2 -17789.135} C_VEL
LIN {X 0,Y 270.192,Z 477.304,A -85,B 0,C 180,E1 -17792.174,E2 -17792.174} C_VEL
LIN {X 0,Y 270.183,Z 477.318,A -85,B 0,C 180,E1 -17795.562,E2 -17795.562} C_VEL
LIN {X 0,Y 270.215,Z 477.296,A -85,B 0,C 180,E1 -17800.236,E2 -17800.236} C_VEL
LIN {X 0,Y 270.335,Z 477.305,A -85,B 0,C 180,E1 -17804.929,E2 -17804.929} C_VEL
LIN {X 0,Y 270.38,Z 477.269,A -85,B 0,C 180,E1 -17809.514,E2 -17809.514} C_VEL
LIN {X 0,Y 270.55,Z 477.257,A -85,B 0,C 180,E1 -17812.535,E2 -17812.535} C_VEL
LIN {X 0,Y 270.764,Z 477.234,A -85,B 0,C 180,E1 -17818.51,E2 -17818.51} C_VEL
LIN {X 0,Y 270.763,Z 477.22,A -85,B 0,C 180,E1 -17821.485,E2 -17821.485} C_VEL
LIN {X 0,Y 270.556,Z 477.27,A -85,B 0,C 180,E1 -17827.46,E2 -17827.46} C_VEL
LIN {X 0,Y 270.381,Z 477.265,A -85,B 0,C 180,E1 -17830.481,E2 -17830.481} C_VEL
LIN {X 0,Y 270.337,Z 477.31,A -85,B 0,C 180,E1 -17835.066,E2 -17835.066} C_VEL
LIN {X 0,Y 270.21,Z 477.29,A -85,B 0,C 180,E1 -17839.76,E2 -17839.76} C_VEL
LIN {X 0,Y 270.176,Z 477.327,A -85,B 0,C 180,E1 -17844.435,E2 -17844.435} C_VEL
LIN {X 0,Y 270.177,Z 477.302,A -85,B 0,C 180,E1 -17847.916,E2 -17847.916} C_VEL
LIN {X 0,Y 270.16,Z 477.334,A -85,B 0,C 180,E1 -17851.348,E2 -17851.348} C_VEL
LIN {X 0,Y 270.187,Z 477.306,A -85,B 0,C 180,E1 -17854.904,E2 -17854.904} C_VEL
LIN {X 0,Y 270.157,Z 477.331,A -85,B 0,C 180,E1 -17858.7,E2 -17858.7} C_VEL
LIN {X 0,Y 270.136,Z 477.336,A -85,B 0,C 180,E1 -17863.243,E2 -17863.243} C_VEL
LIN {X 0,Y 270.118,Z 477.282,A -85,B 0,C 180,E1 -17867.432,E2 -17867.432} C_VEL
LIN {X 0,Y 270.154,Z 477.33,A -85,B 0,C 180,E1 -17871.366,E2 -17871.366} C_VEL
LIN {X 0,Y 270.185,Z 477.292,A -85,B 0,C 180,E1 -17875.092,E2 -17875.092} C_VEL
LIN {X 0,Y 270.207,Z 477.545,A -85,B 0,C 180,E1 -17879.283,E2 -17879.283} C_VEL
LIN {X 0,Y 270.499,Z 478.709,A -85,B 0,C 180,E1 -17879.531,E2 -17879.531} C_VEL
LIN {X 0,Y 282.654,Z 501.214,A -85,B 0,C 180,E1 -17881.634,E2 -17881.634} C_VEL
LIN {X 0,Y 290.758,Z 512.622,A -85,B 0,C 180,E1 -17882.811,E2 -17882.811} C_VEL
LIN {X 0,Y 300.246,Z 523.251,A -85,B 0,C 180,E1 -17884.023,E2 -17884.023} C_VEL
LIN {X 0,Y 307.044,Z 530.171,A -85,B 0,C 180,E1 -17884.892,E2 -17884.892} C_VEL
LIN {X 0,Y 313.803,Z 536.796,A -85,B 0,C 180,E1 -17885.857,E2 -17885.857} C_VEL
LIN {X 0,Y 321.562,Z 543.976,A -85,B 0,C 180,E1 -17887.11,E2 -17887.11} C_VEL
LIN {X 0,Y 329.65,Z 551.27,A -85,B 0,C 180,E1 -17888.615,E2 -17888.615} C_VEL
LIN {X 0,Y 338.592,Z 558.849,A -85,B 0,C 180,E1 -17890.479,E2 -17890.479} C_VEL
LIN {X 0,Y 344.125,Z 563.1,A -85,B 0,C 180,E1 -17891.744,E2 -17891.744} C_VEL
LIN {X 0,Y 350.152,Z 567.875,A -85,B 0,C 180,E1 -17893.242,E2 -17893.242} C_VEL
LIN {X 0,Y 355.209,Z 571.613,A -85,B 0,C 180,E1 -17894.622,E2 -17894.622} C_VEL
LIN {X 0,Y 361.289,Z 576.183,A -85,B 0,C 180,E1 -17896.501,E2 -17896.501} C_VEL
LIN {X 0,Y 366.156,Z 579.077,A -85,B 0,C 180,E1 -17898.195,E2 -17898.195} C_VEL
LIN {X 0,Y 370.704,Z 582.79,A -85,B 0,C 180,E1 -17900.107,E2 -17900.107} C_VEL
LIN {X 0,Y 373.972,Z 585.014,A -85,B 0,C 180,E1 -17901.74,E2 -17901.74} C_VEL
LIN {X 0,Y 377.181,Z 586.834,A -85,B 0,C 180,E1 -17903.733,E2 -17903.733} C_VEL
LIN {X 0,Y 379.028,Z 587.644,A -85,B 0,C 180,E1 -17905.218,E2 -17905.218} C_VEL
LIN {X 0,Y 380.667,Z 588.186,A -85,B 0,C 180,E1 -17907.083,E2 -17907.083} C_VEL
LIN {X 0,Y 381.47,Z 588.727,A -85,B 0,C 180,E1 -17908.944,E2 -17908.944} C_VEL
LIN {X 0,Y 381.613,Z 588.666,A -85,B 0,C 180,E1 -17910,E2 -17910} C_VEL
LIN {X 0,Y 381.22,Z 588.559,A -85,B 0,C 180,E1 -17911.849,E2 -17911.849} C_VEL
LIN {X 0,Y 380.214,Z 587.98,A -85,B 0,C 180,E1 -17913.522,E2 -17913.522} C_VEL
LIN {X 0,Y 378.108,Z 587.279,A -85,B 0,C 180,E1 -17915.578,E2 -17915.578} C_VEL
LIN {X 0,Y 375.238,Z 585.765,A -85,B 0,C 180,E1 -17917.533,E2 -17917.533} C_VEL
LIN {X 0,Y 371.757,Z 583.585,A -85,B 0,C 180,E1 -17919.384,E2 -17919.384} C_VEL
LIN {X 0,Y 367.84,Z 580.437,A -85,B 0,C 180,E1 -17921.134,E2 -17921.134} C_VEL
LIN {X 0,Y 365.676,Z 578.839,A -85,B 0,C 180,E1 -17921.981,E2 -17921.981} C_VEL
LIN {X 0,Y 360.541,Z 575.676,A -85,B 0,C 180,E1 -17923.747,E2 -17923.747} C_VEL
LIN {X 0,Y 354.592,Z 571.101,A -85,B 0,C 180,E1 -17925.549,E2 -17925.549} C_VEL
LIN {X 0,Y 347.443,Z 565.847,A -85,B 0,C 180,E1 -17927.448,E2 -17927.448} C_VEL
LIN {X 0,Y 340.85,Z 560.506,A -85,B 0,C 180,E1 -17929.019,E2 -17929.019} C_VEL
LIN {X 0,Y 334.307,Z 555.291,A -85,B 0,C 180,E1 -17930.435,E2 -17930.435} C_VEL
LIN {X 0,Y 326.063,Z 548.178,A -85,B 0,C 180,E1 -17932.061,E2 -17932.061} C_VEL
LIN {X 0,Y 317.946,Z 540.785,A -85,B 0,C 180,E1 -17933.49,E2 -17933.49} C_VEL
LIN {X 0,Y 308.849,Z 532.114,A -85,B 0,C 180,E1 -17934.861,E2 -17934.861} C_VEL
LIN {X 0,Y 300.464,Z 523.477,A -85,B 0,C 180,E1 -17935.951,E2 -17935.951} C_VEL
LIN {X 0,Y 290.592,Z 512.437,A -85,B 0,C 180,E1 -17937.211,E2 -17937.211} C_VEL
LIN {X 0,Y 282.54,Z 501.029,A -85,B 0,C 180,E1 -17938.384,E2 -17938.384} C_VEL
LIN {X 0,Y 275.528,Z 488.058,A -85,B 0,C 180,E1 -17939.562,E2 -17939.562} C_VEL
LIN {X 0,Y 270.357,Z 478.273,A -85,B 0,C 180,E1 -17940.525,E2 -17940.525} C_VEL
LIN {X 0,Y 270.16,Z 477.393,A -85,B 0,C 180,E1 -17940.861,E2 -17940.861} C_VEL
LIN {X 0,Y 270.185,Z 477.292,A -85,B 0,C 180,E1 -17944.908,E2 -17944.908} C_VEL
LIN {X 0,Y 270.155,Z 477.328,A -85,B 0,C 180,E1 -17948.704,E2 -17948.704} C_VEL
LIN {X 0,Y 270.114,Z 477.288,A -85,B 0,C 180,E1 -17953.242,E2 -17953.242} C_VEL
LIN {X 0,Y 270.139,Z 477.331,A -85,B 0,C 180,E1 -17957.439,E2 -17957.439} C_VEL
LIN {X 0,Y 270.142,Z 477.333,A -85,B 0,C 180,E1 -17961.367,E2 -17961.367} C_VEL
LIN {X 0,Y 270.187,Z 477.306,A -85,B 0,C 180,E1 -17965.096,E2 -17965.096} C_VEL
LIN {X 0,Y 270.162,Z 477.333,A -85,B 0,C 180,E1 -17969.143,E2 -17969.143} C_VEL
LIN {X 0,Y 270.18,Z 477.301,A -85,B 0,C 180,E1 -17972.179,E2 -17972.179} C_VEL
LIN {X 0,Y 270.176,Z 477.327,A -85,B 0,C 180,E1 -17975.565,E2 -17975.565} C_VEL
LIN {X 0,Y 270.21,Z 477.29,A -85,B 0,C 180,E1 -17980.24,E2 -17980.24} C_VEL
LIN {X 0,Y 270.337,Z 477.31,A -85,B 0,C 180,E1 -17984.934,E2 -17984.934} C_VEL
LIN {X 0,Y 270.381,Z 477.265,A -85,B 0,C 180,E1 -17989.519,E2 -17989.519} C_VEL
LIN {X 0,Y 270.556,Z 477.27,A -85,B 0,C 180,E1 -17992.54,E2 -17992.54} C_VEL
LIN {X 0,Y 270.763,Z 477.22,A -85,B 0,C 180,E1 -17998.515,E2 -17998.515} C_VEL
LIN {X 0,Y 270.764,Z 477.234,A -85,B 0,C 180,E1 -18001.49,E2 -18001.49} C_VEL
LIN {X 0,Y 270.55,Z 477.257,A -85,B 0,C 180,E1 -18007.465,E2 -18007.465} C_VEL
LIN {X 0,Y 270.38,Z 477.269,A -85,B 0,C 180,E1 -18010.486,E2 -18010.486} C_VEL
LIN {X 0,Y 270.335,Z 477.305,A -85,B 0,C 180,E1 -18015.071,E2 -18015.071} C_VEL
LIN {X 0,Y 270.215,Z 477.296,A -85,B 0,C 180,E1 -18019.764,E2 -18019.764} C_VEL
LIN {X 0,Y 270.183,Z 477.318,A -85,B 0,C 180,E1 -18024.438,E2 -18024.438} C_VEL
LIN {X 0,Y 270.19,Z 477.305,A -85,B 0,C 180,E1 -18027.92,E2 -18027.92} C_VEL
LIN {X 0,Y 270.176,Z 477.329,A -85,B 0,C 180,E1 -18031.351,E2 -18031.351} C_VEL
LIN {X 0,Y 270.177,Z 477.311,A -85,B 0,C 180,E1 -18032.742,E2 -18032.742} C_VEL
LIN {X 0,Y 269.569,Z 477.387,A -85,B 0,C 180,E1 -18033.987,E2 -18033.987} C_VEL
LIN {X 0,Y 266.743,Z 477.752,A -85,B 0,C 180,E1 -18036.016,E2 -18036.016} C_VEL
LIN {X 0,Y 264.29,Z 478.063,A -85,B 0,C 180,E1 -18037.665,E2 -18037.665} C_VEL
LIN {X 0,Y 263.209,Z 478.187,A -85,B 0,C 180,E1 -18038.943,E2 -18038.943} C_VEL
LIN {X 0,Y 263.108,Z 478.196,A -85,B 0,C 180,E1 -18039.377,E2 -18039.377} C_VEL
LIN {X 0,Y 263.111,Z 478.212,A -85,B 0,C 180,E1 -18041.898,E2 -18041.898} C_VEL
LIN {X 0,Y 263.082,Z 478.216,A -85,B 0,C 180,E1 -18046.163,E2 -18046.163} C_VEL
LIN {X 0,Y 263.076,Z 478.188,A -85,B 0,C 180,E1 -18050.123,E2 -18050.123} C_VEL
LIN {X 0,Y 263.203,Z 478.457,A -85,B 0,C 180,E1 -18051.638,E2 -18051.638} C_VEL
LIN {X 0,Y 264.828,Z 485.76,A -85,B 0,C 180,E1 -18055.357,E2 -18055.357} C_VEL
LIN {X 0,Y 266.311,Z 493.4,A -85,B 0,C 180,E1 -18058.986,E2 -18058.986} C_VEL
LIN {X 0,Y 267.832,Z 497.104,A -85,B 0,C 180,E1 -18059.379,E2 -18059.379} C_VEL
LIN {X 0,Y 272.782,Z 509.22,A -85,B 0,C 180,E1 -18060.347,E2 -18060.347} C_VEL
LIN {X 0,Y 277.912,Z 535.092,A -85,B 0,C 180,E1 -18061.688,E2 -18061.688} C_VEL
LIN {X 0,Y 279.163,Z 544.073,A -85,B 0,C 180,E1 -18062.081,E2 -18062.081} C_VEL
LIN {X 0,Y 277.448,Z 599.834,A -85,B 0,C 180,E1 -18063.534,E2 -18063.534} C_VEL
LIN {X 0,Y 276.705,Z 610.133,A -85,B 0,C 180,E1 -18063.965,E2 -18063.965} C_VEL
LIN {X 0,Y 275.717,Z 619.659,A -85,B 0,C 180,E1 -18064.524,E2 -18064.524} C_VEL
LIN {X 0,Y 274.6,Z 628.752,A -85,B 0,C 180,E1 -18065.223,E2 -18065.223} C_VEL
LIN {X 0,Y 273.234,Z 637.895,A -85,B 0,C 180,E1 -18066.102,E2 -18066.102} C_VEL
LIN {X 0,Y 271.749,Z 646.896,A -85,B 0,C 180,E1 -18067.174,E2 -18067.174} C_VEL
LIN {X 0,Y 270.112,Z 655.621,A -85,B 0,C 180,E1 -18068.438,E2 -18068.438} C_VEL
LIN {X 0,Y 268.616,Z 663.04,A -85,B 0,C 180,E1 -18069.716,E2 -18069.716} C_VEL
LIN {X 0,Y 267.204,Z 670.436,A -85,B 0,C 180,E1 -18071.244,E2 -18071.244} C_VEL
LIN {X 0,Y 265.613,Z 677.829,A -85,B 0,C 180,E1 -18073.079,E2 -18073.079} C_VEL
LIN {X 0,Y 264.251,Z 684.14,A -85,B 0,C 180,E1 -18074.971,E2 -18074.971} C_VEL
LIN {X 0,Y 263.09,Z 689.413,A -85,B 0,C 180,E1 -18076.876,E2 -18076.876} C_VEL
LIN {X 0,Y 262.143,Z 694.51,A -85,B 0,C 180,E1 -18079.183,E2 -18079.183} C_VEL
LIN {X 0,Y 261.523,Z 698.478,A -85,B 0,C 180,E1 -18081.5,E2 -18081.5} C_VEL
LIN {X 0,Y 261.155,Z 701.415,A -85,B 0,C 180,E1 -18083.82,E2 -18083.82} C_VEL
LIN {X 0,Y 261.053,Z 702.918,A -85,B 0,C 180,E1 -18085.368,E2 -18085.368} C_VEL
LIN {X 0,Y 261.09,Z 704.448,A -85,B 0,C 180,E1 -18088.458,E2 -18088.458} C_VEL
LIN {X 0,Y 261.121,Z 704.728,A -85,B 0,C 180,E1 -18090,E2 -18090} C_VEL
LIN {X 0,Y 261.055,Z 703.85,A -85,B 0,C 180,E1 -18093.086,E2 -18093.086} C_VEL
LIN {X 0,Y 261.092,Z 702.451,A -85,B 0,C 180,E1 -18095.137,E2 -18095.137} C_VEL
LIN {X 0,Y 261.523,Z 698.478,A -85,B 0,C 180,E1 -18098.5,E2 -18098.5} C_VEL
LIN {X 0,Y 262.144,Z 694.51,A -85,B 0,C 180,E1 -18100.817,E2 -18100.817} C_VEL
LIN {X 0,Y 263.09,Z 689.413,A -85,B 0,C 180,E1 -18103.124,E2 -18103.124} C_VEL
LIN {X 0,Y 264.814,Z 681.766,A -85,B 0,C 180,E1 -18105.785,E2 -18105.785} C_VEL
LIN {X 0,Y 266.306,Z 674.962,A -85,B 0,C 180,E1 -18107.667,E2 -18107.667} C_VEL
LIN {X 0,Y 267.885,Z 666.865,A -85,B 0,C 180,E1 -18109.515,E2 -18109.515} C_VEL
LIN {X 0,Y 269.465,Z 658.915,A -85,B 0,C 180,E1 -18111.015,E2 -18111.015} C_VEL
LIN {X 0,Y 271.031,Z 650.834,A -85,B 0,C 180,E1 -18112.286,E2 -18112.286} C_VEL
LIN {X 0,Y 272.78,Z 641.077,A -85,B 0,C 180,E1 -18113.537,E2 -18113.537} C_VEL
LIN {X 0,Y 274.087,Z 632.689,A -85,B 0,C 180,E1 -18114.423,E2 -18114.423} C_VEL
LIN {X 0,Y 275.387,Z 622.182,A -85,B 0,C 180,E1 -18115.307,E2 -18115.307} C_VEL
LIN {X 0,Y 276.445,Z 611.851,A -85,B 0,C 180,E1 -18115.96,E2 -18115.96} C_VEL
LIN {X 0,Y 277.405,Z 601.138,A -85,B 0,C 180,E1 -18116.419,E2 -18116.419} C_VEL
LIN {X 0,Y 278.223,Z 577.017,A -85,B 0,C 180,E1 -18117.083,E2 -18117.083} C_VEL
LIN {X 0,Y 279.103,Z 543.055,A -85,B 0,C 180,E1 -18117.954,E2 -18117.954} C_VEL
LIN {X 0,Y 275.665,Z 523.276,A -85,B 0,C 180,E1 -18118.905,E2 -18118.905} C_VEL
LIN {X 0,Y 272.397,Z 507.961,A -85,B 0,C 180,E1 -18119.736,E2 -18119.736} C_VEL
LIN {X 0,Y 266.433,Z 493.802,A -85,B 0,C 180,E1 -18120.932,E2 -18120.932} C_VEL
LIN {X 0,Y 266.155,Z 492.639,A -85,B 0,C 180,E1 -18121.293,E2 -18121.293} C_VEL
LIN {X 0,Y 264.608,Z 484.852,A -85,B 0,C 180,E1 -18125.097,E2 -18125.097} C_VEL
LIN {X 0,Y 263.163,Z 478.298,A -85,B 0,C 180,E1 -18128.487,E2 -18128.487} C_VEL
LIN {X 0,Y 263.077,Z 478.188,A -85,B 0,C 180,E1 -18131.902,E2 -18131.902} C_VEL
LIN {X 0,Y 263.082,Z 478.204,A -85,B 0,C 180,E1 -18136.16,E2 -18136.16} C_VEL
LIN {X 0,Y 263.094,Z 478.198,A -85,B 0,C 180,E1 -18140.123,E2 -18140.123} C_VEL
LIN {X 0,Y 263.158,Z 478.198,A -85,B 0,C 180,E1 -18144.015,E2 -18144.015} C_VEL
LIN {X 0,Y 263.13,Z 478.196,A -85,B 0,C 180,E1 -18147.709,E2 -18147.709} C_VEL
LIN {X 0,Y 263.142,Z 478.185,A -85,B 0,C 180,E1 -18151.806,E2 -18151.806} C_VEL
LIN {X 0,Y 263.116,Z 478.205,A -85,B 0,C 180,E1 -18156.378,E2 -18156.378} C_VEL
LIN {X 0,Y 263.206,Z 478.175,A -85,B 0,C 180,E1 -18159.687,E2 -18159.687} C_VEL
LIN {X 0,Y 263.288,Z 478.178,A -85,B 0,C 180,E1 -18164.516,E2 -18164.516} C_VEL
LIN {X 0,Y 263.324,Z 478.151,A -85,B 0,C 180,E1 -18169.23,E2 -18169.23} C_VEL
LIN {X 0,Y 263.512,Z 478.13,A -85,B 0,C 180,E1 -18172.334,E2 -18172.334} C_VEL
LIN {X 0,Y 263.728,Z 478.11,A -85,B 0,C 180,E1 -18178.471,E2 -18178.471} C_VEL
LIN {X 0,Y 263.727,Z 478.096,A -85,B 0,C 180,E1 -18181.525,E2 -18181.525} C_VEL
LIN {X 0,Y 263.521,Z 478.142,A -85,B 0,C 180,E1 -18187.661,E2 -18187.661} C_VEL
LIN {X 0,Y 263.327,Z 478.145,A -85,B 0,C 180,E1 -18190.765,E2 -18190.765} C_VEL
LIN {X 0,Y 263.284,Z 478.189,A -85,B 0,C 180,E1 -18195.479,E2 -18195.479} C_VEL
LIN {X 0,Y 263.199,Z 478.167,A -85,B 0,C 180,E1 -18200.309,E2 -18200.309} C_VEL
LIN {X 0,Y 263.114,Z 478.199,A -85,B 0,C 180,E1 -18205.298,E2 -18205.298} C_VEL
LIN {X 0,Y 263.11,Z 478.188,A -85,B 0,C 180,E1 -18208.735,E2 -18208.735} C_VEL
LIN {X 0,Y 263.117,Z 478.206,A -85,B 0,C 180,E1 -18212.287,E2 -18212.287} C_VEL
LIN {X 0,Y 263.143,Z 478.192,A -85,B 0,C 180,E1 -18215.982,E2 -18215.982} C_VEL
LIN {X 0,Y 263.061,Z 478.201,A -85,B 0,C 180,E1 -18219.877,E2 -18219.877} C_VEL
LIN {X 0,Y 263.065,Z 478.214,A -85,B 0,C 180,E1 -18223.992,E2 -18223.992} C_VEL
LIN {X 0,Y 263.053,Z 478.16,A -85,B 0,C 180,E1 -18228.42,E2 -18228.42} C_VEL
LIN {X 0,Y 263.102,Z 478.215,A -85,B 0,C 180,E1 -18232.094,E2 -18232.094} C_VEL
LIN {X 0,Y 263.139,Z 478.17,A -85,B 0,C 180,E1 -18235.884,E2 -18235.884} C_VEL
LIN {X 0,Y 263.147,Z 478.43,A -85,B 0,C 180,E1 -18238.402,E2 -18238.402} C_VEL
LIN {X 0,Y 263.522,Z 479.781,A -85,B 0,C 180,E1 -18238.665,E2 -18238.665} C_VEL
LIN {X 0,Y 271.724,Z 494.99,A -85,B 0,C 180,E1 -18240.186,E2 -18240.186} C_VEL
LIN {X 0,Y 277.835,Z 506.079,A -85,B 0,C 180,E1 -18241.232,E2 -18241.232} C_VEL
LIN {X 0,Y 286.343,Z 518.022,A -85,B 0,C 180,E1 -18242.502,E2 -18242.502} C_VEL
LIN {X 0,Y 298.363,Z 531.396,A -85,B 0,C 180,E1 -18244.059,E2 -18244.059} C_VEL
LIN {X 0,Y 308.372,Z 541.136,A -85,B 0,C 180,E1 -18245.331,E2 -18245.331} C_VEL
LIN {X 0,Y 317.152,Z 549.15,A -85,B 0,C 180,E1 -18246.643,E2 -18246.643} C_VEL
LIN {X 0,Y 325.027,Z 556.085,A -85,B 0,C 180,E1 -18248.003,E2 -18248.003} C_VEL
LIN {X 0,Y 332.818,Z 562.664,A -85,B 0,C 180,E1 -18249.52,E2 -18249.52} C_VEL
LIN {X 0,Y 339.215,Z 567.51,A -85,B 0,C 180,E1 -18250.878,E2 -18250.878} C_VEL
LIN {X 0,Y 346.635,Z 573.448,A -85,B 0,C 180,E1 -18252.632,E2 -18252.632} C_VEL
LIN {X 0,Y 352.384,Z 577.545,A -85,B 0,C 180,E1 -18254.137,E2 -18254.137} C_VEL
LIN {X 0,Y 357.571,Z 581.565,A -85,B 0,C 180,E1 -18255.656,E2 -18255.656} C_VEL
LIN {X 0,Y 362.652,Z 584.854,A -85,B 0,C 180,E1 -18257.303,E2 -18257.303} C_VEL
LIN {X 0,Y 366.181,Z 587.049,A -85,B 0,C 180,E1 -18258.575,E2 -18258.575} C_VEL
LIN {X 0,Y 370.333,Z 590.417,A -85,B 0,C 180,E1 -18260.381,E2 -18260.381} C_VEL
LIN {X 0,Y 373.931,Z 592.604,A -85,B 0,C 180,E1 -18262.237,E2 -18262.237} C_VEL
LIN {X 0,Y 377.023,Z 594.25,A -85,B 0,C 180,E1 -18264.27,E2 -18264.27} C_VEL
LIN {X 0,Y 379.071,Z 594.943,A -85,B 0,C 180,E1 -18266.138,E2 -18266.138} C_VEL
LIN {X 0,Y 380.219,Z 595.513,A -85,B 0,C 180,E1 -18267.881,E2 -18267.881} C_VEL
LIN {X 0,Y 380.602,Z 595.773,A -85,B 0,C 180,E1 -18268.942,E2 -18268.942} C_VEL
LIN {X 0,Y 380.75,Z 595.691,A -85,B 0,C 180,E1 -18270,E2 -18270} C_VEL
LIN {X 0,Y 380.431,Z 595.675,A -85,B 0,C 180,E1 -18271.588,E2 -18271.588} C_VEL
LIN {X 0,Y 379.594,Z 595.108,A -85,B 0,C 180,E1 -18273.184,E2 -18273.184} C_VEL
LIN {X 0,Y 377.811,Z 594.59,A -85,B 0,C 180,E1 -18275.067,E2 -18275.067} C_VEL
LIN {X 0,Y 375.046,Z 593.279,A -85,B 0,C 180,E1 -18277.094,E2 -18277.094} C_VEL
LIN {X 0,Y 371.736,Z 591.257,A -85,B 0,C 180,E1 -18278.954,E2 -18278.954} C_VEL
LIN {X 0,Y 368.034,Z 588.637,A -85,B 0,C 180,E1 -18280.656,E2 -18280.656} C_VEL
LIN {X 0,Y 364.288,Z 585.729,A -85,B 0,C 180,E1 -18282.139,E2 -18282.139} C_VEL
LIN {X 0,Y 358.941,Z 582.5,A -85,B 0,C 180,E1 -18283.932,E2 -18283.932} C_VEL
LIN {X 0,Y 353.19,Z 578.223,A -85,B 0,C 180,E1 -18285.636,E2 -18285.636} C_VEL
LIN {X 0,Y 348.298,Z 574.614,A -85,B 0,C 180,E1 -18286.945,E2 -18286.945} C_VEL
LIN {X 0,Y 342.384,Z 570.129,A -85,B 0,C 180,E1 -18288.391,E2 -18288.391} C_VEL
LIN {X 0,Y 335.084,Z 564.484,A -85,B 0,C 180,E1 -18290.012,E2 -18290.012} C_VEL
LIN {X 0,Y 326.549,Z 557.348,A -85,B 0,C 180,E1 -18291.719,E2 -18291.719} C_VEL
LIN {X 0,Y 319.386,Z 551.003,A -85,B 0,C 180,E1 -18292.997,E2 -18292.997} C_VEL
LIN {X 0,Y 312.088,Z 544.534,A -85,B 0,C 180,E1 -18294.142,E2 -18294.142} C_VEL
LIN {X 0,Y 303.771,Z 536.682,A -85,B 0,C 180,E1 -18295.282,E2 -18295.282} C_VEL
LIN {X 0,Y 291.543,Z 524.106,A -85,B 0,C 180,E1 -18296.798,E2 -18296.798} C_VEL
LIN {X 0,Y 284.022,Z 514.925,A -85,B 0,C 180,E1 -18297.831,E2 -18297.831} C_VEL
LIN {X 0,Y 276.665,Z 504.199,A -85,B 0,C 180,E1 -18298.957,E2 -18298.957} C_VEL
LIN {X 0,Y 264.433,Z 481.516,A -85,B 0,C 180,E1 -18301.15,E2 -18301.15} C_VEL
LIN {X 0,Y 263.229,Z 478.851,A -85,B 0,C 180,E1 -18301.479,E2 -18301.479} C_VEL
LIN {X 0,Y 263.113,Z 478.251,A -85,B 0,C 180,E1 -18301.856,E2 -18301.856} C_VEL
LIN {X 0,Y 263.143,Z 478.177,A -85,B 0,C 180,E1 -18305.985,E2 -18305.985} C_VEL
LIN {X 0,Y 263.058,Z 478.181,A -85,B 0,C 180,E1 -18309.881,E2 -18309.881} C_VEL
LIN {X 0,Y 263.059,Z 478.178,A -85,B 0,C 180,E1 -18313.997,E2 -18313.997} C_VEL
LIN {X 0,Y 263.063,Z 478.204,A -85,B 0,C 180,E1 -18318.099,E2 -18318.099} C_VEL
LIN {X 0,Y 263.093,Z 478.216,A -85,B 0,C 180,E1 -18322.095,E2 -18322.095} C_VEL
LIN {X 0,Y 263.142,Z 478.184,A -85,B 0,C 180,E1 -18325.888,E2 -18325.888} C_VEL
LIN {X 0,Y 263.101,Z 478.212,A -85,B 0,C 180,E1 -18329.504,E2 -18329.504} C_VEL
LIN {X 0,Y 263.105,Z 478.182,A -85,B 0,C 180,E1 -18332.996,E2 -18332.996} C_VEL
LIN {X 0,Y 263.109,Z 478.211,A -85,B 0,C 180,E1 -18336.383,E2 -18336.383} C_VEL
LIN {X 0,Y 263.199,Z 478.167,A -85,B 0,C 180,E1 -18339.691,E2 -18339.691} C_VEL
LIN {X 0,Y 263.284,Z 478.189,A -85,B 0,C 180,E1 -18344.521,E2 -18344.521} C_VEL
LIN {X 0,Y 263.327,Z 478.145,A -85,B 0,C 180,E1 -18349.235,E2 -18349.235} C_VEL
LIN {X 0,Y 263.521,Z 478.142,A -85,B 0,C 180,E1 -18352.339,E2 -18352.339} C_VEL
LIN {X 0,Y 263.727,Z 478.096,A -85,B 0,C 180,E1 -18358.475,E2 -18358.475} C_VEL
LIN {X 0,Y 263.728,Z 478.11,A -85,B 0,C 180,E1 -18361.529,E2 -18361.529} C_VEL
LIN {X 0,Y 263.512,Z 478.13,A -85,B 0,C 180,E1 -18367.666,E2 -18367.666} C_VEL
LIN {X 0,Y 263.324,Z 478.151,A -85,B 0,C 180,E1 -18370.77,E2 -18370.77} C_VEL
LIN {X 0,Y 263.288,Z 478.178,A -85,B 0,C 180,E1 -18375.484,E2 -18375.484} C_VEL
LIN {X 0,Y 263.206,Z 478.175,A -85,B 0,C 180,E1 -18380.313,E2 -18380.313} C_VEL
LIN {X 0,Y 263.124,Z 478.193,A -85,B 0,C 180,E1 -18384.752,E2 -18384.752} C_VEL
LIN {X 0,Y 263.131,Z 478.195,A -85,B 0,C 180,E1 -18388.738,E2 -18388.738} C_VEL
LIN {X 0,Y 263.111,Z 478.192,A -85,B 0,C 180,E1 -18392.735,E2 -18392.735} C_VEL
LIN {X 0,Y 263.176,Z 478.202,A -85,B 0,C 180,E1 -18396.762,E2 -18396.762} C_VEL
LIN {X 0,Y 263.108,Z 478.196,A -85,B 0,C 180,E1 -18399.377,E2 -18399.377} C_VEL
LIN {X 0,Y 262.4,Z 478.29,A -85,B 0,C 180,E1 -18400.654,E2 -18400.654} C_VEL
LIN {X 0,Y 259.522,Z 478.657,A -85,B 0,C 180,E1 -18402.736,E2 -18402.736} C_VEL
LIN {X 0,Y 257.109,Z 478.958,A -85,B 0,C 180,E1 -18404.43,E2 -18404.43} C_VEL
LIN {X 0,Y 256.088,Z 479.086,A -85,B 0,C 180,E1 -18405.743,E2 -18405.743} C_VEL
LIN {X 0,Y 256.011,Z 479.091,A -85,B 0,C 180,E1 -18406.188,E2 -18406.188} C_VEL
LIN {X 0,Y 256.095,Z 479.21,A -85,B 0,C 180,E1 -18410.863,E2 -18410.863} C_VEL
LIN {X 0,Y 257.508,Z 485.213,A -85,B 0,C 180,E1 -18414.072,E2 -18414.072} C_VEL
LIN {X 0,Y 259.077,Z 493.073,A -85,B 0,C 180,E1 -18417.991,E2 -18417.991} C_VEL
LIN {X 0,Y 259.766,Z 495.256,A -85,B 0,C 180,E1 -18418.27,E2 -18418.27} C_VEL
LIN {X 0,Y 265.64,Z 508.469,A -85,B 0,C 180,E1 -18419.451,E2 -18419.451} C_VEL
LIN {X 0,Y 267.189,Z 513.19,A -85,B 0,C 180,E1 -18419.789,E2 -18419.789} C_VEL
LIN {X 0,Y 271.794,Z 537.001,A -85,B 0,C 180,E1 -18421.053,E2 -18421.053} C_VEL
LIN {X 0,Y 272.871,Z 544.847,A -85,B 0,C 180,E1 -18421.408,E2 -18421.408} C_VEL
LIN {X 0,Y 271.105,Z 599.688,A -85,B 0,C 180,E1 -18422.867,E2 -18422.867} C_VEL
LIN {X 0,Y 270.346,Z 609.951,A -85,B 0,C 180,E1 -18423.306,E2 -18423.306} C_VEL
LIN {X 0,Y 269.328,Z 619.463,A -85,B 0,C 180,E1 -18423.874,E2 -18423.874} C_VEL
LIN {X 0,Y 268.173,Z 628.556,A -85,B 0,C 180,E1 -18424.587,E2 -18424.587} C_VEL
LIN {X 0,Y 266.764,Z 637.699,A -85,B 0,C 180,E1 -18425.485,E2 -18425.485} C_VEL
LIN {X 0,Y 265.21,Z 646.7,A -85,B 0,C 180,E1 -18426.579,E2 -18426.579} C_VEL
LIN {X 0,Y 263.516,Z 655.424,A -85,B 0,C 180,E1 -18427.87,E2 -18427.87} C_VEL
LIN {X 0,Y 261.965,Z 662.844,A -85,B 0,C 180,E1 -18429.178,E2 -18429.178} C_VEL
LIN {X 0,Y 260.281,Z 670.992,A -85,B 0,C 180,E1 -18430.924,E2 -18430.924} C_VEL
LIN {X 0,Y 258.818,Z 677.633,A -85,B 0,C 180,E1 -18432.621,E2 -18432.621} C_VEL
LIN {X 0,Y 257.391,Z 683.944,A -85,B 0,C 180,E1 -18434.561,E2 -18434.561} C_VEL
LIN {X 0,Y 256.166,Z 689.217,A -85,B 0,C 180,E1 -18436.515,E2 -18436.515} C_VEL
LIN {X 0,Y 255.135,Z 694.313,A -85,B 0,C 180,E1 -18438.883,E2 -18438.883} C_VEL
LIN {X 0,Y 254.48,Z 698.281,A -85,B 0,C 180,E1 -18441.263,E2 -18441.263} C_VEL
LIN {X 0,Y 254.067,Z 701.218,A -85,B 0,C 180,E1 -18443.647,E2 -18443.647} C_VEL
LIN {X 0,Y 253.961,Z 702.722,A -85,B 0,C 180,E1 -18445.238,E2 -18445.238} C_VEL
LIN {X 0,Y 253.998,Z 704.252,A -85,B 0,C 180,E1 -18448.414,E2 -18448.414} C_VEL
LIN {X 0,Y 254.048,Z 704.533,A -85,B 0,C 180,E1 -18450,E2 -18450} C_VEL
LIN {X 0,Y 253.954,Z 703.653,A -85,B 0,C 180,E1 -18453.173,E2 -18453.173} C_VEL
LIN {X 0,Y 253.997,Z 702.488,A -85,B 0,C 180,E1 -18455.039,E2 -18455.039} C_VEL
LIN {X 0,Y 254.309,Z 699.371,A -85,B 0,C 180,E1 -18457.942,E2 -18457.942} C_VEL
LIN {X 0,Y 254.873,Z 695.741,A -85,B 0,C 180,E1 -18460.325,E2 -18460.325} C_VEL
LIN {X 0,Y 255.738,Z 691.006,A -85,B 0,C 180,E1 -18462.7,E2 -18462.7} C_VEL
LIN {X 0,Y 257.097,Z 685.035,A -85,B 0,C 180,E1 -18465.052,E2 -18465.052} C_VEL
LIN {X 0,Y 258.174,Z 680.255,A -85,B 0,C 180,E1 -18466.608,E2 -18466.608} C_VEL
LIN {X 0,Y 259.536,Z 674.766,A -85,B 0,C 180,E1 -18468.144,E2 -18468.144} C_VEL
LIN {X 0,Y 261.181,Z 666.547,A -85,B 0,C 180,E1 -18470.064,E2 -18470.064} C_VEL
LIN {X 0,Y 262.841,Z 658.719,A -85,B 0,C 180,E1 -18471.571,E2 -18471.571} C_VEL
LIN {X 0,Y 264.474,Z 650.638,A -85,B 0,C 180,E1 -18472.869,E2 -18472.869} C_VEL
LIN {X 0,Y 266.279,Z 640.88,A -85,B 0,C 180,E1 -18474.148,E2 -18474.148} C_VEL
LIN {X 0,Y 267.639,Z 632.492,A -85,B 0,C 180,E1 -18475.051,E2 -18475.051} C_VEL
LIN {X 0,Y 268.978,Z 621.986,A -85,B 0,C 180,E1 -18475.954,E2 -18475.954} C_VEL
LIN {X 0,Y 270.08,Z 611.682,A -85,B 0,C 180,E1 -18476.618,E2 -18476.618} C_VEL
LIN {X 0,Y 271.065,Z 601.048,A -85,B 0,C 180,E1 -18477.083,E2 -18477.083} C_VEL
LIN {X 0,Y 271.886,Z 578.165,A -85,B 0,C 180,E1 -18477.728,E2 -18477.728} C_VEL
LIN {X 0,Y 272.858,Z 544.291,A -85,B 0,C 180,E1 -18478.61,E2 -18478.61} C_VEL
LIN {X 0,Y 269.586,Z 525.183,A -85,B 0,C 180,E1 -18479.558,E2 -18479.558} C_VEL
LIN {X 0,Y 266.413,Z 510.384,A -85,B 0,C 180,E1 -18480.394,E2 -18480.394} C_VEL
LIN {X 0,Y 260.437,Z 496.582,A -85,B 0,C 180,E1 -18481.598,E2 -18481.598} C_VEL
LIN {X 0,Y 259.116,Z 493.249,A -85,B 0,C 180,E1 -18481.955,E2 -18481.955} C_VEL
LIN {X 0,Y 257.794,Z 486.783,A -85,B 0,C 180,E1 -18485.126,E2 -18485.126} C_VEL
LIN {X 0,Y 256.511,Z 480.977,A -85,B 0,C 180,E1 -18488.166,E2 -18488.166} C_VEL
LIN {X 0,Y 256.084,Z 479.149,A -85,B 0,C 180,E1 -18489.294,E2 -18489.294} C_VEL
LIN {X 0,Y 256.025,Z 479.089,A -85,B 0,C 180,E1 -18493.334,E2 -18493.334} C_VEL
LIN {X 0,Y 256.059,Z 479.09,A -85,B 0,C 180,E1 -18497.821,E2 -18497.821} C_VEL
LIN {X 0,Y 256.119,Z 479.082,A -85,B 0,C 180,E1 -18502.727,E2 -18502.727} C_VEL
LIN {X 0,Y 256.069,Z 479.064,A -85,B 0,C 180,E1 -18506.705,E2 -18506.705} C_VEL
LIN {X 0,Y 256.055,Z 479.086,A -85,B 0,C 180,E1 -18510.391,E2 -18510.391} C_VEL
LIN {X 0,Y 256.061,Z 479.057,A -85,B 0,C 180,E1 -18513.948,E2 -18513.948} C_VEL
LIN {X 0,Y 256.057,Z 479.087,A -85,B 0,C 180,E1 -18517.4,E2 -18517.4} C_VEL
LIN {X 0,Y 256.098,Z 479.047,A -85,B 0,C 180,E1 -18520.771,E2 -18520.771} C_VEL
LIN {X 0,Y 256.212,Z 479.054,A -85,B 0,C 180,E1 -18524.077,E2 -18524.077} C_VEL
LIN {X 0,Y 256.268,Z 479.033,A -85,B 0,C 180,E1 -18528.93,E2 -18528.93} C_VEL
LIN {X 0,Y 256.454,Z 479.005,A -85,B 0,C 180,E1 -18532.122,E2 -18532.122} C_VEL
LIN {X 0,Y 256.439,Z 479.037,A -85,B 0,C 180,E1 -18536.856,E2 -18536.856} C_VEL
LIN {X 0,Y 256.69,Z 478.986,A -85,B 0,C 180,E1 -18538.429,E2 -18538.429} C_VEL
LIN {X 0,Y 256.689,Z 478.972,A -85,B 0,C 180,E1 -18541.566,E2 -18541.566} C_VEL
LIN {X 0,Y 256.436,Z 479.033,A -85,B 0,C 180,E1 -18546.602,E2 -18546.602} C_VEL
LIN {X 0,Y 256.397,Z 479.007,A -85,B 0,C 180,E1 -18549.463,E2 -18549.463} C_VEL
LIN {X 0,Y 256.205,Z 479.071,A -85,B 0,C 180,E1 -18554.29,E2 -18554.29} C_VEL
LIN {X 0,Y 256.138,Z 479.054,A -85,B 0,C 180,E1 -18557.564,E2 -18557.564} C_VEL
LIN {X 0,Y 256.111,Z 479.06,A -85,B 0,C 180,E1 -18561.094,E2 -18561.094} C_VEL
LIN {X 0,Y 256.076,Z 479.079,A -85,B 0,C 180,E1 -18565.086,E2 -18565.086} C_VEL
LIN {X 0,Y 256.068,Z 479.063,A -85,B 0,C 180,E1 -18568.567,E2 -18568.567} C_VEL
LIN {X 0,Y 256.061,Z 479.091,A -85,B 0,C 180,E1 -18571.697,E2 -18571.697} C_VEL
LIN {X 0,Y 256.068,Z 479.065,A -85,B 0,C 180,E1 -18575.192,E2 -18575.192} C_VEL
LIN {X 0,Y 256.031,Z 479.085,A -85,B 0,C 180,E1 -18579.146,E2 -18579.146} C_VEL
LIN {X 0,Y 256.01,Z 479.096,A -85,B 0,C 180,E1 -18583.334,E2 -18583.334} C_VEL
LIN {X 0,Y 255.99,Z 479.037,A -85,B 0,C 180,E1 -18587.835,E2 -18587.835} C_VEL
LIN {X 0,Y 256.03,Z 479.072,A -85,B 0,C 180,E1 -18590.851,E2 -18590.851} C_VEL
LIN {X 0,Y 256.086,Z 479.077,A -85,B 0,C 180,E1 -18592.86,E2 -18592.86} C_VEL
LIN {X 0,Y 256.064,Z 479.094,A -85,B 0,C 180,E1 -18597.135,E2 -18597.135} C_VEL
LIN {X 0,Y 256.131,Z 479.474,A -85,B 0,C 180,E1 -18597.518,E2 -18597.518} C_VEL
LIN {X 0,Y 256.72,Z 481.256,A -85,B 0,C 180,E1 -18597.786,E2 -18597.786} C_VEL
LIN {X 0,Y 263.319,Z 493.041,A -85,B 0,C 180,E1 -18599.063,E2 -18599.063} C_VEL
LIN {X 0,Y 272.136,Z 509.525,A -85,B 0,C 180,E1 -18600.669,E2 -18600.669} C_VEL
LIN {X 0,Y 280.217,Z 521.191,A -85,B 0,C 180,E1 -18601.933,E2 -18601.933} C_VEL
LIN {X 0,Y 290.655,Z 533.238,A -85,B 0,C 180,E1 -18603.361,E2 -18603.361} C_VEL
LIN {X 0,Y 303.109,Z 545.674,A -85,B 0,C 180,E1 -18604.896,E2 -18604.896} C_VEL
LIN {X 0,Y 312.219,Z 553.849,A -85,B 0,C 180,E1 -18606.134,E2 -18606.134} C_VEL
LIN {X 0,Y 321.362,Z 561.791,A -85,B 0,C 180,E1 -18607.597,E2 -18607.597} C_VEL
LIN {X 0,Y 330.338,Z 569.192,A -85,B 0,C 180,E1 -18609.274,E2 -18609.274} C_VEL
LIN {X 0,Y 338.923,Z 575.729,A -85,B 0,C 180,E1 -18611.083,E2 -18611.083} C_VEL
LIN {X 0,Y 345.899,Z 581.043,A -85,B 0,C 180,E1 -18612.728,E2 -18612.728} C_VEL
LIN {X 0,Y 350.887,Z 584.62,A -85,B 0,C 180,E1 -18614.021,E2 -18614.021} C_VEL
LIN {X 0,Y 356.164,Z 588.543,A -85,B 0,C 180,E1 -18615.541,E2 -18615.541} C_VEL
LIN {X 0,Y 360.923,Z 591.577,A -85,B 0,C 180,E1 -18617.057,E2 -18617.057} C_VEL
LIN {X 0,Y 364.353,Z 593.654,A -85,B 0,C 180,E1 -18618.252,E2 -18618.252} C_VEL
LIN {X 0,Y 368.872,Z 597.168,A -85,B 0,C 180,E1 -18620.127,E2 -18620.127} C_VEL
LIN {X 0,Y 372.361,Z 599.326,A -85,B 0,C 180,E1 -18621.851,E2 -18621.851} C_VEL
LIN {X 0,Y 375.365,Z 600.941,A -85,B 0,C 180,E1 -18623.703,E2 -18623.703} C_VEL
LIN {X 0,Y 377.246,Z 601.73,A -85,B 0,C 180,E1 -18625.195,E2 -18625.195} C_VEL
LIN {X 0,Y 378.895,Z 602.28,A -85,B 0,C 180,E1 -18627.049,E2 -18627.049} C_VEL
LIN {X 0,Y 379.734,Z 602.819,A -85,B 0,C 180,E1 -18628.94,E2 -18628.94} C_VEL
LIN {X 0,Y 379.887,Z 602.717,A -85,B 0,C 180,E1 -18630,E2 -18630} C_VEL
LIN {X 0,Y 379.614,Z 602.721,A -85,B 0,C 180,E1 -18631.43,E2 -18631.43} C_VEL
LIN {X 0,Y 378.718,Z 602.149,A -85,B 0,C 180,E1 -18633.191,E2 -18633.191} C_VEL
LIN {X 0,Y 376.918,Z 601.634,A -85,B 0,C 180,E1 -18635.079,E2 -18635.079} C_VEL
LIN {X 0,Y 374.028,Z 600.281,A -85,B 0,C 180,E1 -18637.175,E2 -18637.175} C_VEL
LIN {X 0,Y 370.773,Z 598.331,A -85,B 0,C 180,E1 -18638.977,E2 -18638.977} C_VEL
LIN {X 0,Y 367.174,Z 595.901,A -85,B 0,C 180,E1 -18640.618,E2 -18640.618} C_VEL
LIN {X 0,Y 362.869,Z 592.609,A -85,B 0,C 180,E1 -18642.301,E2 -18642.301} C_VEL
LIN {X 0,Y 357.467,Z 589.401,A -85,B 0,C 180,E1 -18644.065,E2 -18644.065} C_VEL
LIN {X 0,Y 352.028,Z 585.522,A -85,B 0,C 180,E1 -18645.658,E2 -18645.658} C_VEL
LIN {X 0,Y 347.255,Z 581.911,A -85,B 0,C 180,E1 -18646.93,E2 -18646.93} C_VEL
LIN {X 0,Y 341.277,Z 577.627,A -85,B 0,C 180,E1 -18648.377,E2 -18648.377} C_VEL
LIN {X 0,Y 334.537,Z 572.432,A -85,B 0,C 180,E1 -18649.867,E2 -18649.867} C_VEL
LIN {X 0,Y 327.566,Z 566.851,A -85,B 0,C 180,E1 -18651.273,E2 -18651.273} C_VEL
LIN {X 0,Y 318.993,Z 559.788,A -85,B 0,C 180,E1 -18652.8,E2 -18652.8} C_VEL
LIN {X 0,Y 311.288,Z 553.039,A -85,B 0,C 180,E1 -18654.001,E2 -18654.001} C_VEL
LIN {X 0,Y 302.064,Z 544.701,A -85,B 0,C 180,E1 -18655.239,E2 -18655.239} C_VEL
LIN {X 0,Y 287.882,Z 530.315,A -85,B 0,C 180,E1 -18656.999,E2 -18656.999} C_VEL
LIN {X 0,Y 279.559,Z 520.248,A -85,B 0,C 180,E1 -18658.166,E2 -18658.166} C_VEL
LIN {X 0,Y 271.789,Z 508.955,A -85,B 0,C 180,E1 -18659.39,E2 -18659.39} C_VEL
LIN {X 0,Y 264.859,Z 495.86,A -85,B 0,C 180,E1 -18660.649,E2 -18660.649} C_VEL
LIN {X 0,Y 257.359,Z 482.362,A -85,B 0,C 180,E1 -18662.087,E2 -18662.087} C_VEL
LIN {X 0,Y 256.203,Z 479.765,A -85,B 0,C 180,E1 -18662.412,E2 -18662.412} C_VEL
LIN {X 0,Y 256.073,Z 479.122,A -85,B 0,C 180,E1 -18662.757,E2 -18662.757} C_VEL
LIN {X 0,Y 256.066,Z 479.051,A -85,B 0,C 180,E1 -18665.195,E2 -18665.195} C_VEL
LIN {X 0,Y 256.104,Z 479.078,A -85,B 0,C 180,E1 -18667.272,E2 -18667.272} C_VEL
LIN {X 0,Y 255.991,Z 479.04,A -85,B 0,C 180,E1 -18671.215,E2 -18671.215} C_VEL
LIN {X 0,Y 256.005,Z 479.089,A -85,B 0,C 180,E1 -18675.542,E2 -18675.542} C_VEL
LIN {X 0,Y 255.997,Z 479.078,A -85,B 0,C 180,E1 -18678.789,E2 -18678.789} C_VEL
LIN {X 0,Y 256.089,Z 479.085,A -85,B 0,C 180,E1 -18682.864,E2 -18682.864} C_VEL
LIN {X 0,Y 256.056,Z 479.074,A -85,B 0,C 180,E1 -18686.709,E2 -18686.709} C_VEL
LIN {X 0,Y 256.032,Z 479.083,A -85,B 0,C 180,E1 -18690.393,E2 -18690.393} C_VEL
LIN {X 0,Y 256.059,Z 479.067,A -85,B 0,C 180,E1 -18693.953,E2 -18693.953} C_VEL
LIN {X 0,Y 256.05,Z 479.088,A -85,B 0,C 180,E1 -18697.405,E2 -18697.405} C_VEL
LIN {X 0,Y 256.096,Z 479.046,A -85,B 0,C 180,E1 -18700.776,E2 -18700.776} C_VEL
LIN {X 0,Y 256.207,Z 479.067,A -85,B 0,C 180,E1 -18704.082,E2 -18704.082} C_VEL
LIN {X 0,Y 256.271,Z 479.025,A -85,B 0,C 180,E1 -18708.935,E2 -18708.935} C_VEL
LIN {X 0,Y 256.463,Z 479.018,A -85,B 0,C 180,E1 -18712.127,E2 -18712.127} C_VEL
LIN {X 0,Y 256.438,Z 479.027,A -85,B 0,C 180,E1 -18716.86,E2 -18716.86} C_VEL
LIN {X 0,Y 256.689,Z 478.972,A -85,B 0,C 180,E1 -18718.434,E2 -18718.434} C_VEL
LIN {X 0,Y 256.69,Z 478.986,A -85,B 0,C 180,E1 -18721.571,E2 -18721.571} C_VEL
LIN {X 0,Y 256.448,Z 479.03,A -85,B 0,C 180,E1 -18726.296,E2 -18726.296} C_VEL
LIN {X 0,Y 256.397,Z 479.002,A -85,B 0,C 180,E1 -18729.468,E2 -18729.468} C_VEL
LIN {X 0,Y 256.194,Z 479.069,A -85,B 0,C 180,E1 -18734.296,E2 -18734.296} C_VEL
LIN {X 0,Y 256.139,Z 479.042,A -85,B 0,C 180,E1 -18737.569,E2 -18737.569} C_VEL
LIN {X 0,Y 256.119,Z 479.071,A -85,B 0,C 180,E1 -18741.099,E2 -18741.099} C_VEL
LIN {X 0,Y 256.078,Z 479.064,A -85,B 0,C 180,E1 -18745.087,E2 -18745.087} C_VEL
LIN {X 0,Y 256.087,Z 479.069,A -85,B 0,C 180,E1 -18748.575,E2 -18748.575} C_VEL
LIN {X 0,Y 256.076,Z 479.08,A -85,B 0,C 180,E1 -18751.703,E2 -18751.703} C_VEL
LIN {X 0,Y 256.081,Z 479.069,A -85,B 0,C 180,E1 -18755.195,E2 -18755.195} C_VEL
LIN {X 0,Y 256.068,Z 479.074,A -85,B 0,C 180,E1 -18759.145,E2 -18759.145} C_VEL
LIN {X 0,Y 256.031,Z 479.085,A -85,B 0,C 180,E1 -18763.336,E2 -18763.336} C_VEL
LIN {X 0,Y 256.011,Z 479.091,A -85,B 0,C 180,E1 -18766.188,E2 -18766.188} C_VEL
LIN {X 0,Y 255.305,Z 479.177,A -85,B 0,C 180,E1 -18767.08,E2 -18767.08} C_VEL
LIN {X 0,Y 252.37,Z 479.518,A -85,B 0,C 180,E1 -18768.481,E2 -18768.481} C_VEL
LIN {X 0,Y 249.654,Z 480.125,A -85,B 0,C 180,E1 -18769.881,E2 -18769.881} C_VEL
LIN {X 0,Y 249.263,Z 481.179,A -85,B 0,C 180,E1 -18770.745,E2 -18770.745} C_VEL
LIN {X 0,Y 250.637,Z 486.96,A -85,B 0,C 180,E1 -18773.925,E2 -18773.925} C_VEL
LIN {X 0,Y 251.835,Z 492.929,A -85,B 0,C 180,E1 -18776.981,E2 -18776.981} C_VEL
LIN {X 0,Y 253.364,Z 496.517,A -85,B 0,C 180,E1 -18777.419,E2 -18777.419} C_VEL
LIN {X 0,Y 260.816,Z 513.701,A -85,B 0,C 180,E1 -18778.992,E2 -18778.992} C_VEL
LIN {X 0,Y 264.885,Z 534.17,A -85,B 0,C 180,E1 -18780.144,E2 -18780.144} C_VEL
LIN {X 0,Y 266.627,Z 545.928,A -85,B 0,C 180,E1 -18780.712,E2 -18780.712} C_VEL
LIN {X 0,Y 264.835,Z 598.878,A -85,B 0,C 180,E1 -18782.143,E2 -18782.143} C_VEL
LIN {X 0,Y 264.098,Z 609.112,A -85,B 0,C 180,E1 -18782.582,E2 -18782.582} C_VEL
LIN {X 0,Y 263.1,Z 618.004,A -85,B 0,C 180,E1 -18783.1,E2 -18783.1} C_VEL
LIN {X 0,Y 262.118,Z 626.393,A -85,B 0,C 180,E1 -18783.743,E2 -18783.743} C_VEL
LIN {X 0,Y 260.321,Z 637.503,A -85,B 0,C 180,E1 -18784.836,E2 -18784.836} C_VEL
LIN {X 0,Y 258.691,Z 646.503,A -85,B 0,C 180,E1 -18785.952,E2 -18785.952} C_VEL
LIN {X 0,Y 256.941,Z 655.228,A -85,B 0,C 180,E1 -18787.272,E2 -18787.272} C_VEL
LIN {X 0,Y 255.321,Z 662.647,A -85,B 0,C 180,E1 -18788.61,E2 -18788.61} C_VEL
LIN {X 0,Y 253.747,Z 669.883,A -85,B 0,C 180,E1 -18790.167,E2 -18790.167} C_VEL
LIN {X 0,Y 252.045,Z 677.436,A -85,B 0,C 180,E1 -18792.138,E2 -18792.138} C_VEL
LIN {X 0,Y 250.541,Z 683.747,A -85,B 0,C 180,E1 -18794.128,E2 -18794.128} C_VEL
LIN {X 0,Y 249.229,Z 689.019,A -85,B 0,C 180,E1 -18796.132,E2 -18796.132} C_VEL
LIN {X 0,Y 248.145,Z 694.116,A -85,B 0,C 180,E1 -18798.565,E2 -18798.565} C_VEL
LIN {X 0,Y 247.425,Z 698.084,A -85,B 0,C 180,E1 -18801.012,E2 -18801.012} C_VEL
LIN {X 0,Y 246.989,Z 701.021,A -85,B 0,C 180,E1 -18803.465,E2 -18803.465} C_VEL
LIN {X 0,Y 246.858,Z 702.582,A -85,B 0,C 180,E1 -18805.185,E2 -18805.185} C_VEL
LIN {X 0,Y 246.907,Z 704.056,A -85,B 0,C 180,E1 -18808.369,E2 -18808.369} C_VEL
LIN {X 0,Y 246.978,Z 704.337,A -85,B 0,C 180,E1 -18810,E2 -18810} C_VEL
LIN {X 0,Y 246.858,Z 703.457,A -85,B 0,C 180,E1 -18813.264,E2 -18813.264} C_VEL
LIN {X 0,Y 246.889,Z 702.526,A -85,B 0,C 180,E1 -18814.899,E2 -18814.899} C_VEL
LIN {X 0,Y 247.264,Z 699.174,A -85,B 0,C 180,E1 -18818.17,E2 -18818.17} C_VEL
LIN {X 0,Y 247.856,Z 695.544,A -85,B 0,C 180,E1 -18820.621,E2 -18820.621} C_VEL
LIN {X 0,Y 248.779,Z 690.809,A -85,B 0,C 180,E1 -18823.062,E2 -18823.062} C_VEL
LIN {X 0,Y 250.231,Z 684.839,A -85,B 0,C 180,E1 -18825.475,E2 -18825.475} C_VEL
LIN {X 0,Y 251.677,Z 678.747,A -85,B 0,C 180,E1 -18827.469,E2 -18827.469} C_VEL
LIN {X 0,Y 253.198,Z 672.67,A -85,B 0,C 180,E1 -18829.126,E2 -18829.126} C_VEL
LIN {X 0,Y 254.486,Z 666.349,A -85,B 0,C 180,E1 -18830.616,E2 -18830.616} C_VEL
LIN {X 0,Y 256.229,Z 658.522,A -85,B 0,C 180,E1 -18832.157,E2 -18832.157} C_VEL
LIN {X 0,Y 257.932,Z 650.441,A -85,B 0,C 180,E1 -18833.484,E2 -18833.484} C_VEL
LIN {X 0,Y 259.804,Z 640.684,A -85,B 0,C 180,E1 -18834.79,E2 -18834.79} C_VEL
LIN {X 0,Y 261.226,Z 632.296,A -85,B 0,C 180,E1 -18835.71,E2 -18835.71} C_VEL
LIN {X 0,Y 262.602,Z 621.789,A -85,B 0,C 180,E1 -18836.633,E2 -18836.633} C_VEL
LIN {X 0,Y 263.869,Z 610.793,A -85,B 0,C 180,E1 -18837.339,E2 -18837.339} C_VEL
LIN {X 0,Y 264.81,Z 600.129,A -85,B 0,C 180,E1 -18837.807,E2 -18837.807} C_VEL
LIN {X 0,Y 265.887,Z 569.365,A -85,B 0,C 180,E1 -18838.669,E2 -18838.669} C_VEL
LIN {X 0,Y 266.545,Z 544.747,A -85,B 0,C 180,E1 -18839.333,E2 -18839.333} C_VEL
LIN {X 0,Y 263.317,Z 525.835,A -85,B 0,C 180,E1 -18840.308,E2 -18840.308} C_VEL
LIN {X 0,Y 260.68,Z 513.415,A -85,B 0,C 180,E1 -18841.034,E2 -18841.034} C_VEL
LIN {X 0,Y 255.073,Z 500.351,A -85,B 0,C 180,E1 -18842.213,E2 -18842.213} C_VEL
LIN {X 0,Y 251.952,Z 493.336,A -85,B 0,C 180,E1 -18842.928,E2 -18842.928} C_VEL
LIN {X 0,Y 251.768,Z 492.625,A -85,B 0,C 180,E1 -18843.126,E2 -18843.126} C_VEL
LIN {X 0,Y 250.277,Z 485.189,A -85,B 0,C 180,E1 -18847.03,E2 -18847.03} C_VEL
LIN {X 0,Y 248.992,Z 480.052,A -85,B 0,C 180,E1 -18849.951,E2 -18849.951} C_VEL
LIN {X 0,Y 248.976,Z 479.955,A -85,B 0,C 180,E1 -18852.781,E2 -18852.781} C_VEL
LIN {X 0,Y 248.996,Z 479.968,A -85,B 0,C 180,E1 -18857.356,E2 -18857.356} C_VEL
LIN {X 0,Y 249.046,Z 479.96,A -85,B 0,C 180,E1 -18862.199,E2 -18862.199} C_VEL
LIN {X 0,Y 249.045,Z 479.938,A -85,B 0,C 180,E1 -18865.637,E2 -18865.637} C_VEL
LIN {X 0,Y 249.003,Z 479.968,A -85,B 0,C 180,E1 -18869.464,E2 -18869.464} C_VEL
LIN {X 0,Y 249.013,Z 479.932,A -85,B 0,C 180,E1 -18873.153,E2 -18873.153} C_VEL
LIN {X 0,Y 249.006,Z 479.965,A -85,B 0,C 180,E1 -18876.723,E2 -18876.723} C_VEL
LIN {X 0,Y 249.036,Z 479.931,A -85,B 0,C 180,E1 -18880.203,E2 -18880.203} C_VEL
LIN {X 0,Y 249.158,Z 479.926,A -85,B 0,C 180,E1 -18883.614,E2 -18883.614} C_VEL
LIN {X 0,Y 249.213,Z 479.916,A -85,B 0,C 180,E1 -18888.612,E2 -18888.612} C_VEL
LIN {X 0,Y 249.401,Z 479.88,A -85,B 0,C 180,E1 -18891.898,E2 -18891.898} C_VEL
LIN {X 0,Y 249.251,Z 479.936,A -85,B 0,C 180,E1 -18895.145,E2 -18895.145} C_VEL
LIN {X 0,Y 249.651,Z 479.862,A -85,B 0,C 180,E1 -18898.384,E2 -18898.384} C_VEL
LIN {X 0,Y 249.65,Z 479.848,A -85,B 0,C 180,E1 -18901.611,E2 -18901.611} C_VEL
LIN {X 0,Y 249.413,Z 479.91,A -85,B 0,C 180,E1 -18906.58,E2 -18906.58} C_VEL
LIN {X 0,Y 249.328,Z 479.885,A -85,B 0,C 180,E1 -18909.734,E2 -18909.734} C_VEL
LIN {X 0,Y 249.147,Z 479.95,A -85,B 0,C 180,E1 -18914.704,E2 -18914.704} C_VEL
LIN {X 0,Y 249.07,Z 479.927,A -85,B 0,C 180,E1 -18918.08,E2 -18918.08} C_VEL
LIN {X 0,Y 249.036,Z 479.948,A -85,B 0,C 180,E1 -18921.52,E2 -18921.52} C_VEL
LIN {X 0,Y 249.037,Z 479.949,A -85,B 0,C 180,E1 -18925.438,E2 -18925.438} C_VEL
LIN {X 0,Y 249.016,Z 479.945,A -85,B 0,C 180,E1 -18928.966,E2 -18928.966} C_VEL
LIN {X 0,Y 249.017,Z 479.961,A -85,B 0,C 180,E1 -18932.424,E2 -18932.424} C_VEL
LIN {X 0,Y 249.001,Z 479.957,A -85,B 0,C 180,E1 -18936.347,E2 -18936.347} C_VEL
LIN {X 0,Y 248.961,Z 479.953,A -85,B 0,C 180,E1 -18940.483,E2 -18940.483} C_VEL
LIN {X 0,Y 248.948,Z 479.957,A -85,B 0,C 180,E1 -18944.887,E2 -18944.887} C_VEL
LIN {X 0,Y 248.955,Z 479.914,A -85,B 0,C 180,E1 -18947.35,E2 -18947.35} C_VEL
LIN {X 0,Y 249.027,Z 479.967,A -85,B 0,C 180,E1 -18952.2,E2 -18952.2} C_VEL
LIN {X 0,Y 249.053,Z 480.08,A -85,B 0,C 180,E1 -18956.371,E2 -18956.371} C_VEL
LIN {X 0,Y 249.268,Z 481.143,A -85,B 0,C 180,E1 -18956.668,E2 -18956.668} C_VEL
LIN {X 0,Y 250.804,Z 483.834,A -85,B 0,C 180,E1 -18957.012,E2 -18957.012} C_VEL
LIN {X 0,Y 259.762,Z 500.265,A -85,B 0,C 180,E1 -18958.817,E2 -18958.817} C_VEL
LIN {X 0,Y 267.219,Z 514.182,A -85,B 0,C 180,E1 -18960.211,E2 -18960.211} C_VEL
LIN {X 0,Y 275.165,Z 525.726,A -85,B 0,C 180,E1 -18961.498,E2 -18961.498} C_VEL
LIN {X 0,Y 285.879,Z 538.222,A -85,B 0,C 180,E1 -18963.014,E2 -18963.014} C_VEL
LIN {X 0,Y 299.425,Z 551.676,A -85,B 0,C 180,E1 -18964.691,E2 -18964.691} C_VEL
LIN {X 0,Y 308.968,Z 560.142,A -85,B 0,C 180,E1 -18965.923,E2 -18965.923} C_VEL
LIN {X 0,Y 317.094,Z 567.044,A -85,B 0,C 180,E1 -18967.148,E2 -18967.148} C_VEL
LIN {X 0,Y 324.101,Z 572.688,A -85,B 0,C 180,E1 -18968.348,E2 -18968.348} C_VEL
LIN {X 0,Y 331.067,Z 578.207,A -85,B 0,C 180,E1 -18969.677,E2 -18969.677} C_VEL
LIN {X 0,Y 336.971,Z 582.589,A -85,B 0,C 180,E1 -18970.914,E2 -18970.914} C_VEL
LIN {X 0,Y 344.042,Z 587.828,A -85,B 0,C 180,E1 -18972.541,E2 -18972.541} C_VEL
LIN {X 0,Y 349.928,Z 592.064,A -85,B 0,C 180,E1 -18974.054,E2 -18974.054} C_VEL
LIN {X 0,Y 355.217,Z 595.832,A -85,B 0,C 180,E1 -18975.566,E2 -18975.566} C_VEL
LIN {X 0,Y 359.816,Z 598.642,A -85,B 0,C 180,E1 -18977.016,E2 -18977.016} C_VEL
LIN {X 0,Y 363.067,Z 600.658,A -85,B 0,C 180,E1 -18978.134,E2 -18978.134} C_VEL
LIN {X 0,Y 367.612,Z 604.127,A -85,B 0,C 180,E1 -18980.004,E2 -18980.004} C_VEL
LIN {X 0,Y 371.357,Z 606.343,A -85,B 0,C 180,E1 -18981.829,E2 -18981.829} C_VEL
LIN {X 0,Y 374.369,Z 607.987,A -85,B 0,C 180,E1 -18983.686,E2 -18983.686} C_VEL
LIN {X 0,Y 376.829,Z 608.892,A -85,B 0,C 180,E1 -18985.722,E2 -18985.722} C_VEL
LIN {X 0,Y 378.123,Z 609.398,A -85,B 0,C 180,E1 -18987.337,E2 -18987.337} C_VEL
LIN {X 0,Y 378.765,Z 609.852,A -85,B 0,C 180,E1 -18988.937,E2 -18988.937} C_VEL
LIN {X 0,Y 378.923,Z 609.752,A -85,B 0,C 180,E1 -18990,E2 -18990} C_VEL
LIN {X 0,Y 378.659,Z 609.756,A -85,B 0,C 180,E1 -18991.434,E2 -18991.434} C_VEL
LIN {X 0,Y 377.762,Z 609.19,A -85,B 0,C 180,E1 -18993.199,E2 -18993.199} C_VEL
LIN {X 0,Y 375.943,Z 608.667,A -85,B 0,C 180,E1 -18995.092,E2 -18995.092} C_VEL
LIN {X 0,Y 373.231,Z 607.428,A -85,B 0,C 180,E1 -18997.063,E2 -18997.063} C_VEL
LIN {X 0,Y 369.754,Z 605.401,A -85,B 0,C 180,E1 -18999.002,E2 -18999.002} C_VEL
LIN {X 0,Y 365.969,Z 602.915,A -85,B 0,C 180,E1 -19000.717,E2 -19000.717} C_VEL
LIN {X 0,Y 361.446,Z 599.506,A -85,B 0,C 180,E1 -19002.443,E2 -19002.443} C_VEL
LIN {X 0,Y 356.854,Z 596.855,A -85,B 0,C 180,E1 -19003.941,E2 -19003.941} C_VEL
LIN {X 0,Y 351.734,Z 593.395,A -85,B 0,C 180,E1 -19005.443,E2 -19005.443} C_VEL
LIN {X 0,Y 345.094,Z 588.494,A -85,B 0,C 180,E1 -19007.197,E2 -19007.197} C_VEL
LIN {X 0,Y 338.338,Z 583.678,A -85,B 0,C 180,E1 -19008.78,E2 -19008.78} C_VEL
LIN {X 0,Y 331.068,Z 578.194,A -85,B 0,C 180,E1 -19010.323,E2 -19010.323} C_VEL
LIN {X 0,Y 324.823,Z 573.288,A -85,B 0,C 180,E1 -19011.515,E2 -19011.515} C_VEL
LIN {X 0,Y 317.704,Z 567.532,A -85,B 0,C 180,E1 -19012.755,E2 -19012.755} C_VEL
LIN {X 0,Y 309.716,Z 560.741,A -85,B 0,C 180,E1 -19013.973,E2 -19013.973} C_VEL
LIN {X 0,Y 301.713,Z 553.666,A -85,B 0,C 180,E1 -19015.034,E2 -19015.034} C_VEL
LIN {X 0,Y 289.949,Z 542.533,A -85,B 0,C 180,E1 -19016.457,E2 -19016.457} C_VEL
LIN {X 0,Y 277.266,Z 528.469,A -85,B 0,C 180,E1 -19018.185,E2 -19018.185} C_VEL
LIN {X 0,Y 268.234,Z 515.765,A -85,B 0,C 180,E1 -19019.616,E2 -19019.616} C_VEL
LIN {X 0,Y 262.109,Z 504.909,A -85,B 0,C 180,E1 -19020.725,E2 -19020.725} C_VEL
LIN {X 0,Y 254.285,Z 490.007,A -85,B 0,C 180,E1 -19022.274,E2 -19022.274} C_VEL
LIN {X 0,Y 250.092,Z 482.886,A -85,B 0,C 180,E1 -19023.127,E2 -19023.127} C_VEL
LIN {X 0,Y 249.178,Z 480.743,A -85,B 0,C 180,E1 -19023.399,E2 -19023.399} C_VEL
LIN {X 0,Y 249.018,Z 479.992,A -85,B 0,C 180,E1 -19023.78,E2 -19023.78} C_VEL
LIN {X 0,Y 248.999,Z 479.967,A -85,B 0,C 180,E1 -19028.385,E2 -19028.385} C_VEL
LIN {X 0,Y 248.932,Z 479.918,A -85,B 0,C 180,E1 -19032.778,E2 -19032.778} C_VEL
LIN {X 0,Y 248.965,Z 479.968,A -85,B 0,C 180,E1 -19037.356,E2 -19037.356} C_VEL
LIN {X 0,Y 249.011,Z 479.97,A -85,B 0,C 180,E1 -19042.209,E2 -19042.209} C_VEL
LIN {X 0,Y 249.033,Z 479.94,A -85,B 0,C 180,E1 -19045.641,E2 -19045.641} C_VEL
LIN {X 0,Y 248.985,Z 479.97,A -85,B 0,C 180,E1 -19049.467,E2 -19049.467} C_VEL
LIN {X 0,Y 249.006,Z 479.937,A -85,B 0,C 180,E1 -19053.158,E2 -19053.158} C_VEL
LIN {X 0,Y 248.999,Z 479.968,A -85,B 0,C 180,E1 -19056.728,E2 -19056.728} C_VEL
LIN {X 0,Y 249.032,Z 479.926,A -85,B 0,C 180,E1 -19060.208,E2 -19060.208} C_VEL
LIN {X 0,Y 249.152,Z 479.941,A -85,B 0,C 180,E1 -19063.619,E2 -19063.619} C_VEL
LIN {X 0,Y 249.216,Z 479.906,A -85,B 0,C 180,E1 -19068.618,E2 -19068.618} C_VEL
LIN {X 0,Y 249.409,Z 479.894,A -85,B 0,C 180,E1 -19071.903,E2 -19071.903} C_VEL
LIN {X 0,Y 249.25,Z 479.936,A -85,B 0,C 180,E1 -19075.15,E2 -19075.15} C_VEL
LIN {X 0,Y 249.65,Z 479.848,A -85,B 0,C 180,E1 -19078.389,E2 -19078.389} C_VEL
LIN {X 0,Y 249.651,Z 479.862,A -85,B 0,C 180,E1 -19081.616,E2 -19081.616} C_VEL
LIN {X 0,Y 249.418,Z 479.905,A -85,B 0,C 180,E1 -19086.474,E2 -19086.474} C_VEL
LIN {X 0,Y 249.33,Z 479.883,A -85,B 0,C 180,E1 -19089.739,E2 -19089.739} C_VEL
LIN {X 0,Y 249.141,Z 479.945,A -85,B 0,C 180,E1 -19094.71,E2 -19094.71} C_VEL
LIN {X 0,Y 249.072,Z 479.918,A -85,B 0,C 180,E1 -19098.085,E2 -19098.085} C_VEL
LIN {X 0,Y 249.043,Z 479.955,A -85,B 0,C 180,E1 -19101.524,E2 -19101.524} C_VEL
LIN {X 0,Y 249.04,Z 479.935,A -85,B 0,C 180,E1 -19105.439,E2 -19105.439} C_VEL
LIN {X 0,Y 249.035,Z 479.954,A -85,B 0,C 180,E1 -19108.974,E2 -19108.974} C_VEL
LIN {X 0,Y 249.03,Z 479.949,A -85,B 0,C 180,E1 -19112.428,E2 -19112.428} C_VEL
LIN {X 0,Y 249.016,Z 479.963,A -85,B 0,C 180,E1 -19116.35,E2 -19116.35} C_VEL
LIN {X 0,Y 248.982,Z 479.957,A -85,B 0,C 180,E1 -19120.485,E2 -19120.485} C_VEL
LIN {X 0,Y 248.987,Z 479.968,A -85,B 0,C 180,E1 -19122.788,E2 -19122.788} C_VEL
LIN {X 0,Y 248.971,Z 479.954,A -85,B 0,C 180,E1 -19127.354,E2 -19127.354} C_VEL
LIN {X 0,Y 249.015,Z 480.102,A -85,B 0,C 180,E1 -19130.119,E2 -19130.119} C_VEL
LIN {X 0,Y 249.263,Z 481.179,A -85,B 0,C 180,E1 -19130.745,E2 -19130.745} C_VEL
LIN {X 0,Y 249.003,Z 482.852,A -85,B 0,C 180,E1 -19131.569,E2 -19131.569} C_VEL
LIN {X 0,Y 246.816,Z 486.007,A -85,B 0,C 180,E1 -19132.845,E2 -19132.845} C_VEL
LIN {X 0,Y 244.544,Z 489.172,A -85,B 0,C 180,E1 -19134.143,E2 -19134.143} C_VEL
LIN {X 0,Y 244.191,Z 490.886,A -85,B 0,C 180,E1 -19134.988,E2 -19134.988} C_VEL
LIN {X 0,Y 244.615,Z 492.887,A -85,B 0,C 180,E1 -19135.918,E2 -19135.918} C_VEL
LIN {X 0,Y 246.402,Z 496.832,A -85,B 0,C 180,E1 -19136.397,E2 -19136.397} C_VEL
LIN {X 0,Y 254.3,Z 514.653,A -85,B 0,C 180,E1 -19138.144,E2 -19138.144} C_VEL
LIN {X 0,Y 255.498,Z 518.514,A -85,B 0,C 180,E1 -19138.434,E2 -19138.434} C_VEL
LIN {X 0,Y 259.629,Z 540.671,A -85,B 0,C 180,E1 -19139.685,E2 -19139.685} C_VEL
LIN {X 0,Y 260.426,Z 547.4,A -85,B 0,C 180,E1 -19139.996,E2 -19139.996} C_VEL
LIN {X 0,Y 258.563,Z 599.285,A -85,B 0,C 180,E1 -19141.432,E2 -19141.432} C_VEL
LIN {X 0,Y 257.798,Z 609.121,A -85,B 0,C 180,E1 -19141.866,E2 -19141.866} C_VEL
LIN {X 0,Y 256.784,Z 617.807,A -85,B 0,C 180,E1 -19142.383,E2 -19142.383} C_VEL
LIN {X 0,Y 255.443,Z 628.164,A -85,B 0,C 180,E1 -19143.223,E2 -19143.223} C_VEL
LIN {X 0,Y 253.915,Z 637.307,A -85,B 0,C 180,E1 -19144.155,E2 -19144.155} C_VEL
LIN {X 0,Y 252.21,Z 646.306,A -85,B 0,C 180,E1 -19145.293,E2 -19145.293} C_VEL
LIN {X 0,Y 250.368,Z 655.03,A -85,B 0,C 180,E1 -19146.641,E2 -19146.641} C_VEL
LIN {X 0,Y 248.687,Z 662.45,A -85,B 0,C 180,E1 -19148.01,E2 -19148.01} C_VEL
LIN {X 0,Y 247.054,Z 669.686,A -85,B 0,C 180,E1 -19149.606,E2 -19149.606} C_VEL
LIN {X 0,Y 245.293,Z 677.24,A -85,B 0,C 180,E1 -19151.629,E2 -19151.629} C_VEL
LIN {X 0,Y 243.697,Z 683.55,A -85,B 0,C 180,E1 -19153.669,E2 -19153.669} C_VEL
LIN {X 0,Y 242.309,Z 688.822,A -85,B 0,C 180,E1 -19155.728,E2 -19155.728} C_VEL
LIN {X 0,Y 241.165,Z 693.919,A -85,B 0,C 180,E1 -19158.23,E2 -19158.23} C_VEL
LIN {X 0,Y 240.391,Z 697.887,A -85,B 0,C 180,E1 -19160.747,E2 -19160.747} C_VEL
LIN {X 0,Y 239.914,Z 700.825,A -85,B 0,C 180,E1 -19163.271,E2 -19163.271} C_VEL
LIN {X 0,Y 239.774,Z 702.517,A -85,B 0,C 180,E1 -19165.275,E2 -19165.275} C_VEL
LIN {X 0,Y 239.818,Z 703.86,A -85,B 0,C 180,E1 -19168.321,E2 -19168.321} C_VEL
LIN {X 0,Y 239.886,Z 704.141,A -85,B 0,C 180,E1 -19170,E2 -19170} C_VEL
LIN {X 0,Y 239.764,Z 703.26,A -85,B 0,C 180,E1 -19173.361,E2 -19173.361} C_VEL
LIN {X 0,Y 239.807,Z 702.329,A -85,B 0,C 180,E1 -19175.044,E2 -19175.044} C_VEL
LIN {X 0,Y 240.214,Z 698.977,A -85,B 0,C 180,E1 -19178.412,E2 -19178.412} C_VEL
LIN {X 0,Y 240.857,Z 695.347,A -85,B 0,C 180,E1 -19180.933,E2 -19180.933} C_VEL
LIN {X 0,Y 241.831,Z 690.612,A -85,B 0,C 180,E1 -19183.444,E2 -19183.444} C_VEL
LIN {X 0,Y 243.384,Z 684.642,A -85,B 0,C 180,E1 -19185.922,E2 -19185.922} C_VEL
LIN {X 0,Y 244.908,Z 678.55,A -85,B 0,C 180,E1 -19187.968,E2 -19187.968} C_VEL
LIN {X 0,Y 246.3,Z 673.185,A -85,B 0,C 180,E1 -19189.485,E2 -19189.485} C_VEL
LIN {X 0,Y 247.817,Z 666.15,A -85,B 0,C 180,E1 -19191.197,E2 -19191.197} C_VEL
LIN {X 0,Y 249.659,Z 658.326,A -85,B 0,C 180,E1 -19192.772,E2 -19192.772} C_VEL
LIN {X 0,Y 251.4,Z 650.244,A -85,B 0,C 180,E1 -19194.132,E2 -19194.132} C_VEL
LIN {X 0,Y 253.374,Z 640.487,A -85,B 0,C 180,E1 -19195.463,E2 -19195.463} C_VEL
LIN {X 0,Y 254.851,Z 632.1,A -85,B 0,C 180,E1 -19196.402,E2 -19196.402} C_VEL
LIN {X 0,Y 256.288,Z 621.594,A -85,B 0,C 180,E1 -19197.343,E2 -19197.343} C_VEL
LIN {X 0,Y 257.573,Z 610.777,A -85,B 0,C 180,E1 -19198.054,E2 -19198.054} C_VEL
LIN {X 0,Y 258.512,Z 600.589,A -85,B 0,C 180,E1 -19198.518,E2 -19198.518} C_VEL
LIN {X 0,Y 259.383,Z 577.772,A -85,B 0,C 180,E1 -19199.19,E2 -19199.19} C_VEL
LIN {X 0,Y 260.362,Z 545.842,A -85,B 0,C 180,E1 -19200.061,E2 -19200.061} C_VEL
LIN {X 0,Y 257.403,Z 528.247,A -85,B 0,C 180,E1 -19200.998,E2 -19200.998} C_VEL
LIN {X 0,Y 254.866,Z 516.108,A -85,B 0,C 180,E1 -19201.731,E2 -19201.731} C_VEL
LIN {X 0,Y 248.183,Z 500.563,A -85,B 0,C 180,E1 -19203.206,E2 -19203.206} C_VEL
LIN {X 0,Y 244.682,Z 493.061,A -85,B 0,C 180,E1 -19204.044,E2 -19204.044} C_VEL
LIN {X 0,Y 244.362,Z 491.823,A -85,B 0,C 180,E1 -19204.508,E2 -19204.508} C_VEL
LIN {X 0,Y 243.052,Z 485.621,A -85,B 0,C 180,E1 -19207.97,E2 -19207.97} C_VEL
LIN {X 0,Y 241.934,Z 480.914,A -85,B 0,C 180,E1 -19210.774,E2 -19210.774} C_VEL
LIN {X 0,Y 241.9,Z 480.853,A -85,B 0,C 180,E1 -19214.208,E2 -19214.208} C_VEL
LIN {X 0,Y 241.92,Z 480.851,A -85,B 0,C 180,E1 -19218.071,E2 -19218.071} C_VEL
LIN {X 0,Y 241.987,Z 480.842,A -85,B 0,C 180,E1 -19222.415,E2 -19222.415} C_VEL
LIN {X 0,Y 241.982,Z 480.817,A -85,B 0,C 180,E1 -19226.505,E2 -19226.505} C_VEL
LIN {X 0,Y 241.977,Z 480.838,A -85,B 0,C 180,E1 -19230.611,E2 -19230.611} C_VEL
LIN {X 0,Y 241.997,Z 480.809,A -85,B 0,C 180,E1 -19234.195,E2 -19234.195} C_VEL
LIN {X 0,Y 241.986,Z 480.835,A -85,B 0,C 180,E1 -19238.336,E2 -19238.336} C_VEL
LIN {X 0,Y 242.106,Z 480.798,A -85,B 0,C 180,E1 -19243.322,E2 -19243.322} C_VEL
LIN {X 0,Y 242.147,Z 480.802,A -85,B 0,C 180,E1 -19248.275,E2 -19248.275} C_VEL
LIN {X 0,Y 242.356,Z 480.754,A -85,B 0,C 180,E1 -19251.661,E2 -19251.661} C_VEL
LIN {X 0,Y 242.388,Z 480.775,A -85,B 0,C 180,E1 -19253.337,E2 -19253.337} C_VEL
LIN {X 0,Y 242.611,Z 480.739,A -85,B 0,C 180,E1 -19258.337,E2 -19258.337} C_VEL
LIN {X 0,Y 242.61,Z 480.725,A -85,B 0,C 180,E1 -19261.657,E2 -19261.657} C_VEL
LIN {X 0,Y 242.39,Z 480.786,A -85,B 0,C 180,E1 -19266.657,E2 -19266.657} C_VEL
LIN {X 0,Y 242.256,Z 480.765,A -85,B 0,C 180,E1 -19270.021,E2 -19270.021} C_VEL
LIN {X 0,Y 242.103,Z 480.827,A -85,B 0,C 180,E1 -19275.142,E2 -19275.142} C_VEL
LIN {X 0,Y 242.008,Z 480.801,A -85,B 0,C 180,E1 -19278.626,E2 -19278.626} C_VEL
LIN {X 0,Y 241.966,Z 480.836,A -85,B 0,C 180,E1 -19282.181,E2 -19282.181} C_VEL
LIN {X 0,Y 241.979,Z 480.822,A -85,B 0,C 180,E1 -19285.824,E2 -19285.824} C_VEL
LIN {X 0,Y 241.954,Z 480.834,A -85,B 0,C 180,E1 -19289.587,E2 -19289.587} C_VEL
LIN {X 0,Y 241.969,Z 480.825,A -85,B 0,C 180,E1 -19293.491,E2 -19293.491} C_VEL
LIN {X 0,Y 241.955,Z 480.848,A -85,B 0,C 180,E1 -19297.584,E2 -19297.584} C_VEL
LIN {X 0,Y 241.893,Z 480.84,A -85,B 0,C 180,E1 -19301.928,E2 -19301.928} C_VEL
LIN {X 0,Y 241.876,Z 480.815,A -85,B 0,C 180,E1 -19305.786,E2 -19305.786} C_VEL
LIN {X 0,Y 241.919,Z 480.811,A -85,B 0,C 180,E1 -19310.274,E2 -19310.274} C_VEL
LIN {X 0,Y 241.961,Z 480.808,A -85,B 0,C 180,E1 -19314.485,E2 -19314.485} C_VEL
LIN {X 0,Y 242.047,Z 481.099,A -85,B 0,C 180,E1 -19315.364,E2 -19315.364} C_VEL
LIN {X 0,Y 242.419,Z 482.493,A -85,B 0,C 180,E1 -19315.649,E2 -19315.649} C_VEL
LIN {X 0,Y 250.354,Z 496.344,A -85,B 0,C 180,E1 -19317.364,E2 -19317.364} C_VEL
LIN {X 0,Y 262.11,Z 518.5,A -85,B 0,C 180,E1 -19319.699,E2 -19319.699} C_VEL
LIN {X 0,Y 270.149,Z 530.285,A -85,B 0,C 180,E1 -19321.051,E2 -19321.051} C_VEL
LIN {X 0,Y 280.973,Z 543.071,A -85,B 0,C 180,E1 -19322.636,E2 -19322.636} C_VEL
LIN {X 0,Y 295.27,Z 557.308,A -85,B 0,C 180,E1 -19324.451,E2 -19324.451} C_VEL
LIN {X 0,Y 306.479,Z 567.018,A -85,B 0,C 180,E1 -19325.821,E2 -19325.821} C_VEL
LIN {X 0,Y 315.261,Z 574.356,A -85,B 0,C 180,E1 -19327.105,E2 -19327.105} C_VEL
LIN {X 0,Y 322.966,Z 580.445,A -85,B 0,C 180,E1 -19328.386,E2 -19328.386} C_VEL
LIN {X 0,Y 330.39,Z 585.992,A -85,B 0,C 180,E1 -19329.794,E2 -19329.794} C_VEL
LIN {X 0,Y 338.799,Z 592.313,A -85,B 0,C 180,E1 -19331.593,E2 -19331.593} C_VEL
LIN {X 0,Y 346.153,Z 597.393,A -85,B 0,C 180,E1 -19333.365,E2 -19333.365} C_VEL
LIN {X 0,Y 351.723,Z 601.479,A -85,B 0,C 180,E1 -19334.889,E2 -19334.889} C_VEL
LIN {X 0,Y 357.218,Z 604.964,A -85,B 0,C 180,E1 -19336.538,E2 -19336.538} C_VEL
LIN {X 0,Y 361.052,Z 607.216,A -85,B 0,C 180,E1 -19337.84,E2 -19337.84} C_VEL
LIN {X 0,Y 365.788,Z 610.81,A -85,B 0,C 180,E1 -19339.775,E2 -19339.775} C_VEL
LIN {X 0,Y 369.675,Z 613.152,A -85,B 0,C 180,E1 -19341.643,E2 -19341.643} C_VEL
LIN {X 0,Y 373.051,Z 614.974,A -85,B 0,C 180,E1 -19343.703,E2 -19343.703} C_VEL
LIN {X 0,Y 375.504,Z 615.851,A -85,B 0,C 180,E1 -19345.707,E2 -19345.707} C_VEL
LIN {X 0,Y 376.824,Z 616.359,A -85,B 0,C 180,E1 -19347.328,E2 -19347.328} C_VEL
LIN {X 0,Y 377.431,Z 616.811,A -85,B 0,C 180,E1 -19348.933,E2 -19348.933} C_VEL
LIN {X 0,Y 377.598,Z 616.728,A -85,B 0,C 180,E1 -19350,E2 -19350} C_VEL
LIN {X 0,Y 377.296,Z 616.681,A -85,B 0,C 180,E1 -19351.601,E2 -19351.601} C_VEL
LIN {X 0,Y 376.46,Z 616.172,A -85,B 0,C 180,E1 -19353.211,E2 -19353.211} C_VEL
LIN {X 0,Y 374.595,Z 615.617,A -85,B 0,C 180,E1 -19355.111,E2 -19355.111} C_VEL
LIN {X 0,Y 371.857,Z 614.382,A -85,B 0,C 180,E1 -19357.089,E2 -19357.089} C_VEL
LIN {X 0,Y 368.32,Z 612.381,A -85,B 0,C 180,E1 -19359.037,E2 -19359.037} C_VEL
LIN {X 0,Y 364.302,Z 609.752,A -85,B 0,C 180,E1 -19360.858,E2 -19360.858} C_VEL
LIN {X 0,Y 359.676,Z 606.27,A -85,B 0,C 180,E1 -19362.649,E2 -19362.649} C_VEL
LIN {X 0,Y 354.306,Z 603.157,A -85,B 0,C 180,E1 -19364.368,E2 -19364.368} C_VEL
LIN {X 0,Y 347.964,Z 598.771,A -85,B 0,C 180,E1 -19366.168,E2 -19366.168} C_VEL
LIN {X 0,Y 341.998,Z 594.489,A -85,B 0,C 180,E1 -19367.666,E2 -19367.666} C_VEL
LIN {X 0,Y 335.382,Z 589.74,A -85,B 0,C 180,E1 -19369.163,E2 -19369.163} C_VEL
LIN {X 0,Y 328.665,Z 584.758,A -85,B 0,C 180,E1 -19370.547,E2 -19370.547} C_VEL
LIN {X 0,Y 321.87,Z 579.545,A -85,B 0,C 180,E1 -19371.806,E2 -19371.806} C_VEL
LIN {X 0,Y 312.743,Z 572.31,A -85,B 0,C 180,E1 -19373.292,E2 -19373.292} C_VEL
LIN {X 0,Y 303.082,Z 564.197,A -85,B 0,C 180,E1 -19374.612,E2 -19374.612} C_VEL
LIN {X 0,Y 290.442,Z 552.706,A -85,B 0,C 180,E1 -19376.133,E2 -19376.133} C_VEL
LIN {X 0,Y 277.567,Z 539.302,A -85,B 0,C 180,E1 -19377.84,E2 -19377.84} C_VEL
LIN {X 0,Y 269.67,Z 529.565,A -85,B 0,C 180,E1 -19379.028,E2 -19379.028} C_VEL
LIN {X 0,Y 261.926,Z 518.171,A -85,B 0,C 180,E1 -19380.335,E2 -19380.335} C_VEL
LIN {X 0,Y 255.472,Z 506.108,A -85,B 0,C 180,E1 -19381.582,E2 -19381.582} C_VEL
LIN {X 0,Y 247.663,Z 491.518,A -85,B 0,C 180,E1 -19383.203,E2 -19383.203} C_VEL
LIN {X 0,Y 243.17,Z 483.925,A -85,B 0,C 180,E1 -19384.169,E2 -19384.169} C_VEL
LIN {X 0,Y 242.09,Z 481.423,A -85,B 0,C 180,E1 -19384.533,E2 -19384.533} C_VEL
LIN {X 0,Y 241.989,Z 480.853,A -85,B 0,C 180,E1 -19384.938,E2 -19384.938} C_VEL
LIN {X 0,Y 241.972,Z 480.841,A -85,B 0,C 180,E1 -19388.358,E2 -19388.358} C_VEL
LIN {X 0,Y 241.872,Z 480.802,A -85,B 0,C 180,E1 -19393.418,E2 -19393.418} C_VEL
LIN {X 0,Y 241.887,Z 480.855,A -85,B 0,C 180,E1 -19396.582,E2 -19396.582} C_VEL
LIN {X 0,Y 241.964,Z 480.845,A -85,B 0,C 180,E1 -19401.649,E2 -19401.649} C_VEL
LIN {X 0,Y 241.964,Z 480.823,A -85,B 0,C 180,E1 -19404.489,E2 -19404.489} C_VEL
LIN {X 0,Y 241.94,Z 480.85,A -85,B 0,C 180,E1 -19408.478,E2 -19408.478} C_VEL
LIN {X 0,Y 241.943,Z 480.815,A -85,B 0,C 180,E1 -19412.308,E2 -19412.308} C_VEL
LIN {X 0,Y 241.974,Z 480.844,A -85,B 0,C 180,E1 -19416.01,E2 -19416.01} C_VEL
LIN {X 0,Y 241.974,Z 480.809,A -85,B 0,C 180,E1 -19419.605,E2 -19419.605} C_VEL
LIN {X 0,Y 242.1,Z 480.817,A -85,B 0,C 180,E1 -19423.327,E2 -19423.327} C_VEL
LIN {X 0,Y 242.151,Z 480.789,A -85,B 0,C 180,E1 -19428.281,E2 -19428.281} C_VEL
LIN {X 0,Y 242.363,Z 480.766,A -85,B 0,C 180,E1 -19431.666,E2 -19431.666} C_VEL
LIN {X 0,Y 242.39,Z 480.786,A -85,B 0,C 180,E1 -19433.343,E2 -19433.343} C_VEL
LIN {X 0,Y 242.61,Z 480.725,A -85,B 0,C 180,E1 -19438.343,E2 -19438.343} C_VEL
LIN {X 0,Y 242.611,Z 480.739,A -85,B 0,C 180,E1 -19441.663,E2 -19441.663} C_VEL
LIN {X 0,Y 242.388,Z 480.775,A -85,B 0,C 180,E1 -19446.663,E2 -19446.663} C_VEL
LIN {X 0,Y 242.258,Z 480.764,A -85,B 0,C 180,E1 -19450.027,E2 -19450.027} C_VEL
LIN {X 0,Y 242.101,Z 480.82,A -85,B 0,C 180,E1 -19455.147,E2 -19455.147} C_VEL
LIN {X 0,Y 242.011,Z 480.797,A -85,B 0,C 180,E1 -19458.631,E2 -19458.631} C_VEL
LIN {X 0,Y 241.973,Z 480.841,A -85,B 0,C 180,E1 -19462.186,E2 -19462.186} C_VEL
LIN {X 0,Y 241.987,Z 480.81,A -85,B 0,C 180,E1 -19465.829,E2 -19465.829} C_VEL
LIN {X 0,Y 241.97,Z 480.84,A -85,B 0,C 180,E1 -19469.591,E2 -19469.591} C_VEL
LIN {X 0,Y 241.982,Z 480.817,A -85,B 0,C 180,E1 -19473.495,E2 -19473.495} C_VEL
LIN {X 0,Y 241.987,Z 480.842,A -85,B 0,C 180,E1 -19477.585,E2 -19477.585} C_VEL
LIN {X 0,Y 241.92,Z 480.851,A -85,B 0,C 180,E1 -19481.929,E2 -19481.929} C_VEL
LIN {X 0,Y 241.897,Z 480.849,A -85,B 0,C 180,E1 -19486.584,E2 -19486.584} C_VEL
LIN {X 0,Y 241.964,Z 481.007,A -85,B 0,C 180,E1 -19489.342,E2 -19489.342} C_VEL
LIN {X 0,Y 243.637,Z 487.986,A -85,B 0,C 180,E1 -19493.381,E2 -19493.381} C_VEL
LIN {X 0,Y 244.191,Z 490.886,A -85,B 0,C 180,E1 -19494.988,E2 -19494.988} C_VEL
LIN {X 0,Y 244.811,Z 493.009,A -85,B 0,C 180,E1 -19495.699,E2 -19495.699} C_VEL
LIN {X 0,Y 245.815,Z 495.96,A -85,B 0,C 180,E1 -19496.212,E2 -19496.212} C_VEL
LIN {X 0,Y 247.438,Z 501.269,A -85,B 0,C 180,E1 -19496.705,E2 -19496.705} C_VEL
LIN {X 0,Y 248.412,Z 507.309,A -85,B 0,C 180,E1 -19497.042,E2 -19497.042} C_VEL
LIN {X 0,Y 249.476,Z 519.936,A -85,B 0,C 180,E1 -19497.634,E2 -19497.634} C_VEL
LIN {X 0,Y 253.641,Z 542.723,A -85,B 0,C 180,E1 -19498.963,E2 -19498.963} C_VEL
LIN {X 0,Y 254.262,Z 548.205,A -85,B 0,C 180,E1 -19499.223,E2 -19499.223} C_VEL
LIN {X 0,Y 252.382,Z 598.559,A -85,B 0,C 180,E1 -19500.641,E2 -19500.641} C_VEL
LIN {X 0,Y 251.588,Z 608.341,A -85,B 0,C 180,E1 -19501.069,E2 -19501.069} C_VEL
LIN {X 0,Y 250.524,Z 617.611,A -85,B 0,C 180,E1 -19501.631,E2 -19501.631} C_VEL
LIN {X 0,Y 249.121,Z 627.968,A -85,B 0,C 180,E1 -19502.487,E2 -19502.487} C_VEL
LIN {X 0,Y 247.547,Z 637.111,A -85,B 0,C 180,E1 -19503.439,E2 -19503.439} C_VEL
LIN {X 0,Y 245.77,Z 646.11,A -85,B 0,C 180,E1 -19504.6,E2 -19504.6} C_VEL
LIN {X 0,Y 243.871,Z 654.834,A -85,B 0,C 180,E1 -19505.98,E2 -19505.98} C_VEL
LIN {X 0,Y 242.101,Z 662.253,A -85,B 0,C 180,E1 -19507.379,E2 -19507.379} C_VEL
LIN {X 0,Y 240.376,Z 669.489,A -85,B 0,C 180,E1 -19509.013,E2 -19509.013} C_VEL
LIN {X 0,Y 238.541,Z 677.043,A -85,B 0,C 180,E1 -19511.09,E2 -19511.09} C_VEL
LIN {X 0,Y 236.863,Z 683.353,A -85,B 0,C 180,E1 -19513.185,E2 -19513.185} C_VEL
LIN {X 0,Y 235.406,Z 688.625,A -85,B 0,C 180,E1 -19515.3,E2 -19515.3} C_VEL
LIN {X 0,Y 234.178,Z 693.721,A -85,B 0,C 180,E1 -19517.873,E2 -19517.873} C_VEL
LIN {X 0,Y 233.374,Z 697.69,A -85,B 0,C 180,E1 -19520.466,E2 -19520.466} C_VEL
LIN {X 0,Y 232.837,Z 700.628,A -85,B 0,C 180,E1 -19523.065,E2 -19523.065} C_VEL
LIN {X 0,Y 232.686,Z 702.456,A -85,B 0,C 180,E1 -19525.386,E2 -19525.386} C_VEL
LIN {X 0,Y 232.731,Z 703.664,A -85,B 0,C 180,E1 -19528.27,E2 -19528.27} C_VEL
LIN {X 0,Y 232.797,Z 703.945,A -85,B 0,C 180,E1 -19530,E2 -19530} C_VEL
LIN {X 0,Y 232.675,Z 703.064,A -85,B 0,C 180,E1 -19533.463,E2 -19533.463} C_VEL
LIN {X 0,Y 232.736,Z 702.133,A -85,B 0,C 180,E1 -19535.198,E2 -19535.198} C_VEL
LIN {X 0,Y 233.182,Z 698.781,A -85,B 0,C 180,E1 -19538.667,E2 -19538.667} C_VEL
LIN {X 0,Y 233.874,Z 695.151,A -85,B 0,C 180,E1 -19541.264,E2 -19541.264} C_VEL
LIN {X 0,Y 234.896,Z 690.414,A -85,B 0,C 180,E1 -19543.848,E2 -19543.848} C_VEL
LIN {X 0,Y 236.552,Z 684.445,A -85,B 0,C 180,E1 -19546.394,E2 -19546.394} C_VEL
LIN {X 0,Y 238.155,Z 678.354,A -85,B 0,C 180,E1 -19548.496,E2 -19548.496} C_VEL
LIN {X 0,Y 239.728,Z 672.245,A -85,B 0,C 180,E1 -19550.255,E2 -19550.255} C_VEL
LIN {X 0,Y 241.195,Z 665.953,A -85,B 0,C 180,E1 -19551.809,E2 -19551.809} C_VEL
LIN {X 0,Y 243.097,Z 658.128,A -85,B 0,C 180,E1 -19553.423,E2 -19553.423} C_VEL
LIN {X 0,Y 244.908,Z 650.047,A -85,B 0,C 180,E1 -19554.814,E2 -19554.814} C_VEL
LIN {X 0,Y 246.982,Z 640.291,A -85,B 0,C 180,E1 -19556.171,E2 -19556.171} C_VEL
LIN {X 0,Y 248.507,Z 631.904,A -85,B 0,C 180,E1 -19557.131,E2 -19557.131} C_VEL
LIN {X 0,Y 250.013,Z 621.398,A -85,B 0,C 180,E1 -19558.089,E2 -19558.089} C_VEL
LIN {X 0,Y 251.324,Z 610.754,A -85,B 0,C 180,E1 -19558.804,E2 -19558.804} C_VEL
LIN {X 0,Y 252.255,Z 601.024,A -85,B 0,C 180,E1 -19559.265,E2 -19559.265} C_VEL
LIN {X 0,Y 253.096,Z 580.529,A -85,B 0,C 180,E1 -19559.893,E2 -19559.893} C_VEL
LIN {X 0,Y 254.2,Z 546.657,A -85,B 0,C 180,E1 -19560.835,E2 -19560.835} C_VEL
LIN {X 0,Y 250.526,Z 525.401,A -85,B 0,C 180,E1 -19562.034,E2 -19562.034} C_VEL
LIN {X 0,Y 249.007,Z 518.577,A -85,B 0,C 180,E1 -19562.479,E2 -19562.479} C_VEL
LIN {X 0,Y 242.566,Z 503.708,A -85,B 0,C 180,E1 -19563.963,E2 -19563.963} C_VEL
LIN {X 0,Y 237.381,Z 492.78,A -85,B 0,C 180,E1 -19565.25,E2 -19565.25} C_VEL
LIN {X 0,Y 236.882,Z 490.393,A -85,B 0,C 180,E1 -19566.396,E2 -19566.396} C_VEL
LIN {X 0,Y 235.365,Z 483.873,A -85,B 0,C 180,E1 -19570.277,E2 -19570.277} C_VEL
LIN {X 0,Y 234.861,Z 481.779,A -85,B 0,C 180,E1 -19571.681,E2 -19571.681} C_VEL
LIN {X 0,Y 234.871,Z 481.717,A -85,B 0,C 180,E1 -19575.901,E2 -19575.901} C_VEL
LIN {X 0,Y 234.862,Z 481.722,A -85,B 0,C 180,E1 -19578.825,E2 -19578.825} C_VEL
LIN {X 0,Y 234.922,Z 481.708,A -85,B 0,C 180,E1 -19581.077,E2 -19581.077} C_VEL
LIN {X 0,Y 234.905,Z 481.7,A -85,B 0,C 180,E1 -19585.355,E2 -19585.355} C_VEL
LIN {X 0,Y 234.956,Z 481.698,A -85,B 0,C 180,E1 -19587.421,E2 -19587.421} C_VEL
LIN {X 0,Y 234.897,Z 481.707,A -85,B 0,C 180,E1 -19591.396,E2 -19591.396} C_VEL
LIN {X 0,Y 234.899,Z 481.704,A -85,B 0,C 180,E1 -19595.234,E2 -19595.234} C_VEL
LIN {X 0,Y 234.935,Z 481.705,A -85,B 0,C 180,E1 -19598.96,E2 -19598.96} C_VEL
LIN {X 0,Y 235.05,Z 481.673,A -85,B 0,C 180,E1 -19603.096,E2 -19603.096} C_VEL
LIN {X 0,Y 235.079,Z 481.685,A -85,B 0,C 180,E1 -19607.918,E2 -19607.918} C_VEL
LIN {X 0,Y 235.294,Z 481.631,A -85,B 0,C 180,E1 -19611.409,E2 -19611.409} C_VEL
LIN {X 0,Y 235.339,Z 481.648,A -85,B 0,C 180,E1 -19613.137,E2 -19613.137} C_VEL
LIN {X 0,Y 235.57,Z 481.615,A -85,B 0,C 180,E1 -19618.288,E2 -19618.288} C_VEL
LIN {X 0,Y 235.569,Z 481.601,A -85,B 0,C 180,E1 -19621.707,E2 -19621.707} C_VEL
LIN {X 0,Y 235.342,Z 481.663,A -85,B 0,C 180,E1 -19626.858,E2 -19626.858} C_VEL
LIN {X 0,Y 235.18,Z 481.645,A -85,B 0,C 180,E1 -19630.326,E2 -19630.326} C_VEL
LIN {X 0,Y 235.054,Z 481.704,A -85,B 0,C 180,E1 -19635.608,E2 -19635.608} C_VEL
LIN {X 0,Y 234.95,Z 481.678,A -85,B 0,C 180,E1 -19639.207,E2 -19639.207} C_VEL
LIN {X 0,Y 234.909,Z 481.723,A -85,B 0,C 180,E1 -19642.885,E2 -19642.885} C_VEL
LIN {X 0,Y 234.897,Z 481.695,A -85,B 0,C 180,E1 -19646.663,E2 -19646.663} C_VEL
LIN {X 0,Y 234.886,Z 481.726,A -85,B 0,C 180,E1 -19650.571,E2 -19650.571} C_VEL
LIN {X 0,Y 234.931,Z 481.705,A -85,B 0,C 180,E1 -19653.111,E2 -19653.111} C_VEL
LIN {X 0,Y 234.896,Z 481.718,A -85,B 0,C 180,E1 -19656.751,E2 -19656.751} C_VEL
LIN {X 0,Y 234.902,Z 481.718,A -85,B 0,C 180,E1 -19658.933,E2 -19658.933} C_VEL
LIN {X 0,Y 234.84,Z 481.734,A -85,B 0,C 180,E1 -19663.493,E2 -19663.493} C_VEL
LIN {X 0,Y 234.825,Z 481.68,A -85,B 0,C 180,E1 -19666.5,E2 -19666.5} C_VEL
LIN {X 0,Y 234.906,Z 481.702,A -85,B 0,C 180,E1 -19671.077,E2 -19671.077} C_VEL
LIN {X 0,Y 234.953,Z 481.959,A -85,B 0,C 180,E1 -19674.161,E2 -19674.161} C_VEL
LIN {X 0,Y 235.223,Z 483.031,A -85,B 0,C 180,E1 -19674.446,E2 -19674.446} C_VEL
LIN {X 0,Y 236.895,Z 485.772,A -85,B 0,C 180,E1 -19674.854,E2 -19674.854} C_VEL
LIN {X 0,Y 246.655,Z 502.941,A -85,B 0,C 180,E1 -19677.033,E2 -19677.033} C_VEL
LIN {X 0,Y 256.351,Z 521.704,A -85,B 0,C 180,E1 -19679.041,E2 -19679.041} C_VEL
LIN {X 0,Y 263.636,Z 532.694,A -85,B 0,C 180,E1 -19680.332,E2 -19680.332} C_VEL
LIN {X 0,Y 270.719,Z 541.758,A -85,B 0,C 180,E1 -19681.458,E2 -19681.458} C_VEL
LIN {X 0,Y 282.808,Z 554.946,A -85,B 0,C 180,E1 -19683.162,E2 -19683.162} C_VEL
LIN {X 0,Y 294.12,Z 565.484,A -85,B 0,C 180,E1 -19684.56,E2 -19684.56} C_VEL
LIN {X 0,Y 303.251,Z 573.307,A -85,B 0,C 180,E1 -19685.65,E2 -19685.65} C_VEL
LIN {X 0,Y 313.026,Z 581.297,A -85,B 0,C 180,E1 -19686.996,E2 -19686.996} C_VEL
LIN {X 0,Y 321.585,Z 587.965,A -85,B 0,C 180,E1 -19688.418,E2 -19688.418} C_VEL
LIN {X 0,Y 329.504,Z 593.649,A -85,B 0,C 180,E1 -19689.923,E2 -19689.923} C_VEL
LIN {X 0,Y 336.829,Z 599.201,A -85,B 0,C 180,E1 -19691.507,E2 -19691.507} C_VEL
LIN {X 0,Y 343.751,Z 603.971,A -85,B 0,C 180,E1 -19693.171,E2 -19693.171} C_VEL
LIN {X 0,Y 349.807,Z 608.337,A -85,B 0,C 180,E1 -19694.817,E2 -19694.817} C_VEL
LIN {X 0,Y 355.743,Z 612.008,A -85,B 0,C 180,E1 -19696.619,E2 -19696.619} C_VEL
LIN {X 0,Y 359.081,Z 614.059,A -85,B 0,C 180,E1 -19697.772,E2 -19697.772} C_VEL
LIN {X 0,Y 363.614,Z 617.476,A -85,B 0,C 180,E1 -19699.623,E2 -19699.623} C_VEL
LIN {X 0,Y 366.919,Z 619.529,A -85,B 0,C 180,E1 -19701.186,E2 -19701.186} C_VEL
LIN {X 0,Y 369.062,Z 620.7,A -85,B 0,C 180,E1 -19702.34,E2 -19702.34} C_VEL
LIN {X 0,Y 370.845,Z 621.652,A -85,B 0,C 180,E1 -19703.471,E2 -19703.471} C_VEL
LIN {X 0,Y 372.373,Z 622.29,A -85,B 0,C 180,E1 -19704.585,E2 -19704.585} C_VEL
LIN {X 0,Y 373.639,Z 622.697,A -85,B 0,C 180,E1 -19705.685,E2 -19705.685} C_VEL
LIN {X 0,Y 374.607,Z 623.003,A -85,B 0,C 180,E1 -19706.774,E2 -19706.774} C_VEL
LIN {X 0,Y 375.233,Z 623.398,A -85,B 0,C 180,E1 -19707.853,E2 -19707.853} C_VEL
LIN {X 0,Y 375.595,Z 623.668,A -85,B 0,C 180,E1 -19708.928,E2 -19708.928} C_VEL
LIN {X 0,Y 375.772,Z 623.581,A -85,B 0,C 180,E1 -19710,E2 -19710} C_VEL
LIN {X 0,Y 375.617,Z 623.605,A -85,B 0,C 180,E1 -19711.072,E2 -19711.072} C_VEL
LIN {X 0,Y 375.241,Z 623.39,A -85,B 0,C 180,E1 -19712.147,E2 -19712.147} C_VEL
LIN {X 0,Y 374.618,Z 623.001,A -85,B 0,C 180,E1 -19713.226,E2 -19713.226} C_VEL
LIN {X 0,Y 373.567,Z 622.713,A -85,B 0,C 180,E1 -19714.396,E2 -19714.396} C_VEL
LIN {X 0,Y 372.391,Z 622.311,A -85,B 0,C 180,E1 -19715.415,E2 -19715.415} C_VEL
LIN {X 0,Y 370.879,Z 621.615,A -85,B 0,C 180,E1 -19716.528,E2 -19716.528} C_VEL
LIN {X 0,Y 368.823,Z 620.643,A -85,B 0,C 180,E1 -19717.766,E2 -19717.766} C_VEL
LIN {X 0,Y 365.348,Z 618.609,A -85,B 0,C 180,E1 -19719.584,E2 -19719.584} C_VEL
LIN {X 0,Y 361.034,Z 615.62,A -85,B 0,C 180,E1 -19721.455,E2 -19721.455} C_VEL
LIN {X 0,Y 357.426,Z 612.931,A -85,B 0,C 180,E1 -19722.818,E2 -19722.818} C_VEL
LIN {X 0,Y 352.195,Z 609.873,A -85,B 0,C 180,E1 -19724.487,E2 -19724.487} C_VEL
LIN {X 0,Y 346.223,Z 605.822,A -85,B 0,C 180,E1 -19726.182,E2 -19726.182} C_VEL
LIN {X 0,Y 339.617,Z 601.089,A -85,B 0,C 180,E1 -19727.848,E2 -19727.848} C_VEL
LIN {X 0,Y 332.78,Z 596.228,A -85,B 0,C 180,E1 -19729.388,E2 -19729.388} C_VEL
LIN {X 0,Y 326.722,Z 591.755,A -85,B 0,C 180,E1 -19730.624,E2 -19730.624} C_VEL
LIN {X 0,Y 318.798,Z 585.797,A -85,B 0,C 180,E1 -19732.072,E2 -19732.072} C_VEL
LIN {X 0,Y 310.879,Z 579.616,A -85,B 0,C 180,E1 -19733.313,E2 -19733.313} C_VEL
LIN {X 0,Y 302.127,Z 572.423,A -85,B 0,C 180,E1 -19734.485,E2 -19734.485} C_VEL
LIN {X 0,Y 289.8,Z 561.723,A -85,B 0,C 180,E1 -19735.952,E2 -19735.952} C_VEL
LIN {X 0,Y 275.27,Z 547.013,A -85,B 0,C 180,E1 -19737.871,E2 -19737.871} C_VEL
LIN {X 0,Y 265.564,Z 535.38,A -85,B 0,C 180,E1 -19739.347,E2 -19739.347} C_VEL
LIN {X 0,Y 257.032,Z 522.838,A -85,B 0,C 180,E1 -19740.831,E2 -19740.831} C_VEL
LIN {X 0,Y 250.194,Z 510.014,A -85,B 0,C 180,E1 -19742.203,E2 -19742.203} C_VEL
LIN {X 0,Y 242.723,Z 495.843,A -85,B 0,C 180,E1 -19743.824,E2 -19743.824} C_VEL
LIN {X 0,Y 236.543,Z 485.391,A -85,B 0,C 180,E1 -19745.221,E2 -19745.221} C_VEL
LIN {X 0,Y 235.078,Z 482.535,A -85,B 0,C 180,E1 -19745.641,E2 -19745.641} C_VEL
LIN {X 0,Y 234.921,Z 481.773,A -85,B 0,C 180,E1 -19746.026,E2 -19746.026} C_VEL
LIN {X 0,Y 234.9,Z 481.703,A -85,B 0,C 180,E1 -19748.937,E2 -19748.937} C_VEL
LIN {X 0,Y 234.825,Z 481.68,A -85,B 0,C 180,E1 -19753.5,E2 -19753.5} C_VEL
LIN {X 0,Y 234.84,Z 481.734,A -85,B 0,C 180,E1 -19756.507,E2 -19756.507} C_VEL
LIN {X 0,Y 234.908,Z 481.718,A -85,B 0,C 180,E1 -19761.081,E2 -19761.081} C_VEL
LIN {X 0,Y 234.892,Z 481.7,A -85,B 0,C 180,E1 -19765.359,E2 -19765.359} C_VEL
LIN {X 0,Y 234.943,Z 481.712,A -85,B 0,C 180,E1 -19767.426,E2 -19767.426} C_VEL
LIN {X 0,Y 234.882,Z 481.699,A -85,B 0,C 180,E1 -19771.4,E2 -19771.4} C_VEL
LIN {X 0,Y 234.907,Z 481.719,A -85,B 0,C 180,E1 -19775.241,E2 -19775.241} C_VEL
LIN {X 0,Y 234.928,Z 481.694,A -85,B 0,C 180,E1 -19778.965,E2 -19778.965} C_VEL
LIN {X 0,Y 235.044,Z 481.69,A -85,B 0,C 180,E1 -19783.1,E2 -19783.1} C_VEL
LIN {X 0,Y 235.083,Z 481.674,A -85,B 0,C 180,E1 -19787.923,E2 -19787.923} C_VEL
LIN {X 0,Y 235.299,Z 481.641,A -85,B 0,C 180,E1 -19791.414,E2 -19791.414} C_VEL
LIN {X 0,Y 235.342,Z 481.663,A -85,B 0,C 180,E1 -19793.142,E2 -19793.142} C_VEL
LIN {X 0,Y 235.569,Z 481.601,A -85,B 0,C 180,E1 -19798.293,E2 -19798.293} C_VEL
LIN {X 0,Y 235.57,Z 481.615,A -85,B 0,C 180,E1 -19801.712,E2 -19801.712} C_VEL
LIN {X 0,Y 235.339,Z 481.648,A -85,B 0,C 180,E1 -19806.863,E2 -19806.863} C_VEL
LIN {X 0,Y 235.182,Z 481.647,A -85,B 0,C 180,E1 -19810.331,E2 -19810.331} C_VEL
LIN {X 0,Y 235.039,Z 481.693,A -85,B 0,C 180,E1 -19815.614,E2 -19815.614} C_VEL
LIN {X 0,Y 234.954,Z 481.678,A -85,B 0,C 180,E1 -19819.213,E2 -19819.213} C_VEL
LIN {X 0,Y 234.908,Z 481.721,A -85,B 0,C 180,E1 -19822.891,E2 -19822.891} C_VEL
LIN {X 0,Y 234.908,Z 481.688,A -85,B 0,C 180,E1 -19826.667,E2 -19826.667} C_VEL
LIN {X 0,Y 234.901,Z 481.725,A -85,B 0,C 180,E1 -19830.575,E2 -19830.575} C_VEL
LIN {X 0,Y 234.944,Z 481.695,A -85,B 0,C 180,E1 -19833.116,E2 -19833.116} C_VEL
LIN {X 0,Y 234.919,Z 481.723,A -85,B 0,C 180,E1 -19836.753,E2 -19836.753} C_VEL
LIN {X 0,Y 234.916,Z 481.709,A -85,B 0,C 180,E1 -19838.937,E2 -19838.937} C_VEL
LIN {X 0,Y 234.865,Z 481.72,A -85,B 0,C 180,E1 -19843.494,E2 -19843.494} C_VEL
LIN {X 0,Y 234.859,Z 481.715,A -85,B 0,C 180,E1 -19848.063,E2 -19848.063} C_VEL
LIN {X 0,Y 234.88,Z 481.827,A -85,B 0,C 180,E1 -19848.424,E2 -19848.424} C_VEL
LIN {X 0,Y 236.473,Z 488.379,A -85,B 0,C 180,E1 -19852.429,E2 -19852.429} C_VEL
LIN {X 0,Y 237.329,Z 492.543,A -85,B 0,C 180,E1 -19854.699,E2 -19854.699} C_VEL
LIN {X 0,Y 239.084,Z 496.434,A -85,B 0,C 180,E1 -19855.218,E2 -19855.218} C_VEL
LIN {X 0,Y 246.398,Z 512.267,A -85,B 0,C 180,E1 -19856.922,E2 -19856.922} C_VEL
LIN {X 0,Y 249.476,Z 519.936,A -85,B 0,C 180,E1 -19857.634,E2 -19857.634} C_VEL
LIN {X 0,Y 249.918,Z 527.693,A -85,B 0,C 180,E1 -19857.955,E2 -19857.955} C_VEL
LIN {X 0,Y 249.475,Z 535.557,A -85,B 0,C 180,E1 -19858.153,E2 -19858.153} C_VEL
LIN {X 0,Y 248.055,Z 551.394,A -85,B 0,C 180,E1 -19858.478,E2 -19858.478} C_VEL
LIN {X 0,Y 246.17,Z 599.017,A -85,B 0,C 180,E1 -19859.855,E2 -19859.855} C_VEL
LIN {X 0,Y 245.315,Z 609.154,A -85,B 0,C 180,E1 -19860.325,E2 -19860.325} C_VEL
LIN {X 0,Y 244.13,Z 618.677,A -85,B 0,C 180,E1 -19860.936,E2 -19860.936} C_VEL
LIN {X 0,Y 242.851,Z 627.772,A -85,B 0,C 180,E1 -19861.714,E2 -19861.714} C_VEL
LIN {X 0,Y 241.219,Z 636.915,A -85,B 0,C 180,E1 -19862.685,E2 -19862.685} C_VEL
LIN {X 0,Y 239.379,Z 645.914,A -85,B 0,C 180,E1 -19863.872,E2 -19863.872} C_VEL
LIN {X 0,Y 237.402,Z 654.638,A -85,B 0,C 180,E1 -19865.282,E2 -19865.282} C_VEL
LIN {X 0,Y 235.554,Z 662.057,A -85,B 0,C 180,E1 -19866.714,E2 -19866.714} C_VEL
LIN {X 0,Y 233.711,Z 669.291,A -85,B 0,C 180,E1 -19868.385,E2 -19868.385} C_VEL
LIN {X 0,Y 231.816,Z 676.846,A -85,B 0,C 180,E1 -19870.52,E2 -19870.52} C_VEL
LIN {X 0,Y 230.024,Z 683.156,A -85,B 0,C 180,E1 -19872.669,E2 -19872.669} C_VEL
LIN {X 0,Y 228.523,Z 688.428,A -85,B 0,C 180,E1 -19874.846,E2 -19874.846} C_VEL
LIN {X 0,Y 227.211,Z 693.524,A -85,B 0,C 180,E1 -19877.495,E2 -19877.495} C_VEL
LIN {X 0,Y 226.339,Z 697.493,A -85,B 0,C 180,E1 -19880.167,E2 -19880.167} C_VEL
LIN {X 0,Y 225.786,Z 700.431,A -85,B 0,C 180,E1 -19882.848,E2 -19882.848} C_VEL
LIN {X 0,Y 225.579,Z 702.426,A -85,B 0,C 180,E1 -19885.566,E2 -19885.566} C_VEL
LIN {X 0,Y 225.627,Z 703.467,A -85,B 0,C 180,E1 -19888.215,E2 -19888.215} C_VEL
LIN {X 0,Y 225.71,Z 703.75,A -85,B 0,C 180,E1 -19890,E2 -19890} C_VEL
LIN {X 0,Y 225.588,Z 702.868,A -85,B 0,C 180,E1 -19893.572,E2 -19893.572} C_VEL
LIN {X 0,Y 225.65,Z 701.936,A -85,B 0,C 180,E1 -19895.361,E2 -19895.361} C_VEL
LIN {X 0,Y 226.142,Z 698.584,A -85,B 0,C 180,E1 -19898.939,E2 -19898.939} C_VEL
LIN {X 0,Y 226.88,Z 694.953,A -85,B 0,C 180,E1 -19901.616,E2 -19901.616} C_VEL
LIN {X 0,Y 227.98,Z 690.217,A -85,B 0,C 180,E1 -19904.277,E2 -19904.277} C_VEL
LIN {X 0,Y 229.733,Z 684.249,A -85,B 0,C 180,E1 -19906.895,E2 -19906.895} C_VEL
LIN {X 0,Y 231.022,Z 679.468,A -85,B 0,C 180,E1 -19908.628,E2 -19908.628} C_VEL
LIN {X 0,Y 232.535,Z 674.22,A -85,B 0,C 180,E1 -19910.267,E2 -19910.267} C_VEL
LIN {X 0,Y 234.589,Z 665.756,A -85,B 0,C 180,E1 -19912.456,E2 -19912.456} C_VEL
LIN {X 0,Y 236.603,Z 657.932,A -85,B 0,C 180,E1 -19914.106,E2 -19914.106} C_VEL
LIN {X 0,Y 238.49,Z 649.851,A -85,B 0,C 180,E1 -19915.53,E2 -19915.53} C_VEL
LIN {X 0,Y 240.626,Z 640.095,A -85,B 0,C 180,E1 -19916.917,E2 -19916.917} C_VEL
LIN {X 0,Y 242.216,Z 631.708,A -85,B 0,C 180,E1 -19917.896,E2 -19917.896} C_VEL
LIN {X 0,Y 243.766,Z 621.201,A -85,B 0,C 180,E1 -19918.876,E2 -19918.876} C_VEL
LIN {X 0,Y 245.117,Z 610.722,A -85,B 0,C 180,E1 -19919.594,E2 -19919.594} C_VEL
